"A_1113_MXZ11_O1"	Q 24.2	BOOL	// ASPIRATION FAN TANK 3
"A_1114_MXZ11_O1"	Q 24.3	BOOL	// ASPIRATION FAN TANK 4
"A_1115_MXZ11_O1"	Q 24.4	BOOL	// ASPIRATION FAN TANK 5
"A_1116_MXZ11_O1"	Q 24.5	BOOL	// ASPIRATION FAN TANK 6
"A_1117_MXZ11_O1"	Q 24.6	BOOL	// ASPIRATION FAN TANK 7
"A_1118_MXZ11_O1"	Q 24.7	BOOL	// ASPIRATION FAN TANK 8
"A_1119_MXZ11_O1"	Q 25.0	BOOL	// ASPIRATION FAN TANK 9
"A_1120_MXZ11_O1"	Q 25.1	BOOL	// ASPIRATION FAN TANK 10
"A_1121_MXZ11_O1"	Q 25.2	BOOL	// ASPIRATION FAN TANK 11
"A_1122_MXZ11_O1"	Q 25.3	BOOL	// ASPIRATION FAN TANK 12
"A_1123_MXZ11_O1"	Q 25.4	BOOL	// ASPIRATION FAN TANK 13
"A_1124_MXZ11_O1"	Q 25.5	BOOL	// ASPIRATION FAN TANK 14
"A_1125_MXZ11_O1"	Q 25.6	BOOL	// ASPIRATION FAN TANK 15
"A_1126_MXZ11_O1"	Q 25.7	BOOL	// ASPIRATION FAN TANK 16
"A_1127_MXZ11_O1"	Q 26.0	BOOL	// ASPIRATION FAN TANK 17
"A_1127_MXZ21_O1"	Q 26.1	BOOL	// DISCHARGE SLIDE T17 CLOSED
"A_1127_MXZ21_O2"	Q 26.2	BOOL	// DISCHARGE SLIDE T17 OPENED
"A_1128_MXZ11_O1"	Q 26.3	BOOL	// ASPIRATION FAN TANK 18
"A_1128_MXZ21_O1"	Q 26.4	BOOL	// DISCHARGE SLIDE T18 CLOSED
"A_1128_MXZ21_O2"	Q 26.5	BOOL	// DISCHARGE SLIDE T18 OPENED
"A_1129_MXZ11_O1"	Q 26.6	BOOL	// ASPIRATION FAN TANK 19
"A_1129_MXZ21_O1"	Q 26.7	BOOL	// DISCHARGE SLIDE T19 CLOSED
"A_1129_MXZ21_O2"	Q 27.0	BOOL	// DISCHARGE SLIDE T19 OPENED
"A_1130_MXZ11_O1"	Q 27.1	BOOL	// ASPIRATION FAN TANK 20
"A_1130_MXZ21_O1"	Q 27.2	BOOL	// DISCHARGE SLIDE T20 CLOSED
"A_1130_MXZ21_O2"	Q 27.3	BOOL	// DISCHARGE SLIDE T20 OPENED
"A_1131_MXZ11_O1"	Q 27.4	BOOL	// ASPIRATION FAN TANK 21
"A_1131_MXZ21_O1"	Q 27.5	BOOL	// DISCHARGE SLIDE T21 CLOSED
"A_1131_MXZ21_O2"	Q 27.6	BOOL	// DISCHARGE SLIDE T21 OPENED
"A_1132_MXZ11_O1"	Q 27.7	BOOL	// ASPIRATION FAN TANK 22
"A_1132_MXZ21_O1"	Q 28.0	BOOL	// DISCHARGE SLIDE T22 CLOSED
"A_1132_MXZ21_O2"	Q 28.1	BOOL	// DISCHARGE SLIDE T22 OPENED
"A_1133_MXZ11_O1"	Q 28.2	BOOL	// ASPIRATION FAN TANK 23
"A_1133_MXZ21_O1"	Q 28.3	BOOL	// DISCHARGE SLIDE T23 CLOSED
"A_1133_MXZ21_O2"	Q 28.4	BOOL	// DISCHARGE SLIDE T23 OPENED
"A_1134_MXZ11_O1"	Q 28.5	BOOL	// ASPIRATION FAN TANK 24
"A_1134_MXZ21_O1"	Q 28.6	BOOL	// DISCHARGE SLIDE T24 CLOSED
"A_1134_MXZ21_O2"	Q 28.7	BOOL	// DISCHARGE SLIDE T24 OPENED
"A_1151_MXZ11_O1"	Q 29.0	BOOL	// COMPRESSED AIR GROUP S1-S4
"A_1152_MXZ11_O1"	Q 29.1	BOOL	// COMPRESSED AIR GROUP S5-S8
"A_1153_MXZ11_O1"	Q 29.2	BOOL	// COMPRESSED AIR GROUP S9-S12
"A_1154_MXZ11_O1"	Q 29.3	BOOL	// COMPRESSED AIR GROUP S13-S16
"A_1155_MXZ11_O1"	Q 29.4	BOOL	// COMPRESSED AIR GROUP S17-S20
"A_1156_MXZ11_O1"	Q 29.5	BOOL	// COMPRESSED AIR GROUP S21-S24
"A_1111_QXV42_O2"	Q 32.1	BOOL	// BALL VALVE FRESH-AIR TANK 1
"A_1112_QXV42_O2"	Q 32.3	BOOL	// BALL VALVE FRESH-AIR TANK 2
"A_1113_QXV42_O2"	Q 32.5	BOOL	// BALL VALVE FRESH-AIR TANK 3
"A_1114_QXV42_O2"	Q 32.7	BOOL	// BALL VALVE FRESH-AIR TANK 4
"A_1115_QXV42_O2"	Q 33.1	BOOL	// BALL VALVE FRESH-AIR TANK 5
"A_1116_QXV42_O2"	Q 33.3	BOOL	// BALL VALVE FRESH-AIR TANK 6
"A_1117_QXV42_O2"	Q 33.5	BOOL	// BALL VALVE FRESH-AIR TANK 7
"A_1118_QXV42_O2"	Q 33.7	BOOL	// BALL VALVE FRESH-AIR TANK 8
"A_1119_QXV42_O2"	Q 34.1	BOOL	// BALL VALVE FRESH-AIR TANK 9
"A_1120_QXV42_O2"	Q 34.3	BOOL	// BALL VALVE FRESH-AIR TANK 10
"A_1121_QXV42_O2"	Q 34.5	BOOL	// BALL VALVE FRESH-AIR TANK 11
"A_1122_QXV42_O2"	Q 34.7	BOOL	// BALL VALVE FRESH-AIR TANK 12
"A_1123_QXV42_O2"	Q 44.1	BOOL	// BALL VALVE FRESH-AIR TANK 13
"A_1124_QXV42_O2"	Q 44.3	BOOL	// BALL VALVE FRESH-AIR TANK 14
"A_1125_QXV42_O2"	Q 44.5	BOOL	// BALL VALVE FRESH-AIR TANK 15
"A_1126_QXV42_O2"	Q 44.7	BOOL	// BALL VALVE FRESH-AIR TANK 16
"A_1127_QXV42_O2"	Q 45.1	BOOL	// BALL VALVE FRESH-AIR TANK 17
"A_1128_QXV42_O2"	Q 45.3	BOOL	// BALL VALVE FRESH-AIR TANK 18
"A_1129_QXV42_O2"	Q 45.5	BOOL	// BALL VALVE FRESH-AIR TANK 19
"A_1130_QXV42_O2"	Q 45.7	BOOL	// BALL VALVE FRESH-AIR TANK 20
"A_1131_QXV42_O2"	Q 46.1	BOOL	// BALL VALVE FRESH-AIR TANK 21
"A_1132_QXV42_O2"	Q 46.3	BOOL	// BALL VALVE FRESH-AIR TANK 22
"A_1133_QXV42_O2"	Q 46.5	BOOL	// BALL VALVE FRESH-AIR TANK 23
"A_1134_QXV42_O2"	Q 46.7	BOOL	// BALL VALVE FRESH-AIR TANK 24
"A_1161_MXZ01_O1"	Q 48.0	BOOL	// SLIDE GATE 1 - CO2 OPEN
"A_1161_MXZ01_O2"	Q 48.1	BOOL	// SLIDE GATE 1 - CO2 CLOSE
"A_1162_MXZ01_O1"	Q 48.2	BOOL	// SLIDE GATE 2 - CO2 OPEN
"A_1162_MXZ01_O2"	Q 48.3	BOOL	// SLIDE GATE 2 - CO2 CLOSE
"A_1163_MXZ01_O1"	Q 48.4	BOOL	// SLIDE GATE 3 - CO2 OPEN
"A_1163_MXZ01_O2"	Q 48.5	BOOL	// SLIDE GATE 3 - CO2 CLOSE
"A_1164_MXZ01_O1"	Q 48.6	BOOL	// SLIDE GATE 4 - CO2 OPEN
"A_1164_MXZ01_O2"	Q 48.7	BOOL	// SLIDE GATE 4 - CO2 CLOSE
"A_1165_MXZ01_O1"	Q 49.0	BOOL	// SLIDE GATE 5 - CO2 OPEN
"A_1165_MXZ01_O2"	Q 49.1	BOOL	// SLIDE GATE 5 - CO2 CLOSE
"A_1166_MXZ01_O1"	Q 49.2	BOOL	// SLIDE GATE 6 - CO2 OPEN
"A_1166_MXZ01_O2"	Q 49.3	BOOL	// SLIDE GATE 6 - CO2 CLOSE
"A_1167_MXZ01_O1"	Q 49.4	BOOL	// SLIDE GATE 7 - CO2 OPEN
"A_1167_MXZ01_O2"	Q 49.5	BOOL	// SLIDE GATE 7 - CO2 CLOSE
"A_1168_MXZ01_O1"	Q 49.6	BOOL	// SLIDE GATE 8 - CO2 OPEN
"A_1168_MXZ01_O2"	Q 49.7	BOOL	// SLIDE GATE 8 - CO2 CLOSE
"A_1169_MXZ01_O1"	Q 50.0	BOOL	// SLIDE GATE 9 - CO2 OPEN
"A_1169_MXZ01_O2"	Q 50.1	BOOL	// SLIDE GATE 9 - CO2 CLOSE
"A_1170_MXZ01_O1"	Q 50.2	BOOL	// SLIDE GATE 10-CO2 OPEN
"A_1170_MXZ01_O2"	Q 50.3	BOOL	// SLIDE GATE 10-CO2 CLOSE
"A_1171_MXZ01_O1"	Q 50.4	BOOL	// SLIDE GATE 11-CO2 OPEN
"A_1171_MXZ01_O2"	Q 50.5	BOOL	// SLIDE GATE 11-CO2 CLOSE
"A_1172_MXZ01_O1"	Q 50.6	BOOL	// SLIDE GATE 12-CO2 OPEN
"A_1172_MXZ01_O2"	Q 50.7	BOOL	// SLIDE GATE 12-CO2 CLOSE
"A_1173_MXZ01_O1"	Q 51.0	BOOL	// SLIDE GATE 13-CO2 OPEN
"A_1173_MXZ01_O2"	Q 51.1	BOOL	// SLIDE GATE 13-CO2 CLOSE
"A_1174_MXZ01_O1"	Q 51.2	BOOL	// SLIDE GATE 14-CO2 OPEN
"A_1174_MXZ01_O2"	Q 51.3	BOOL	// SLIDE GATE 14-CO2 CLOSE
"A_1175_MXZ01_O1"	Q 51.4	BOOL	// SLIDE GATE 15-CO2 OPEN
"A_1175_MXZ01_O2"	Q 51.5	BOOL	// SLIDE GATE 15-CO2 CLOSE
"A_1176_MXZ01_O1"	Q 51.6	BOOL	// SLIDE GATE 16-CO2 OPEN
"A_1176_MXZ01_O2"	Q 51.7	BOOL	// SLIDE GATE 16-CO2 CLOSE
"A_1177_MXZ01_O1"	Q 52.0	BOOL	// SLIDE GATE 17-CO2 OPEN
"A_1177_MXZ01_O2"	Q 52.1	BOOL	// SLIDE GATE 17-CO2 CLOSE
"A_1178_MXZ01_O1"	Q 52.2	BOOL	// SLIDE GATE 18-CO2 OPEN
"A_1178_MXZ01_O2"	Q 52.3	BOOL	// SLIDE GATE 18-CO2 CLOSE
"A_1179_MXZ01_O1"	Q 52.4	BOOL	// SLIDE GATE 19-CO2 OPEN
"A_1179_MXZ01_O2"	Q 52.5	BOOL	// SLIDE GATE 19-CO2 CLOSE
"A_1180_MXZ01_O1"	Q 52.6	BOOL	// SLIDE GATE 20-CO2 OPEN
"A_1180_MXZ01_O2"	Q 52.7	BOOL	// SLIDE GATE 20-CO2 CLOSE
"A_1181_MXZ01_O1"	Q 53.0	BOOL	// SLIDE GATE 21-CO2 OPEN
"A_1181_MXZ01_O2"	Q 53.1	BOOL	// SLIDE GATE 21-CO2 CLOSE
"A_1182_MXZ01_O1"	Q 53.2	BOOL	// SLIDE GATE 22-CO2 OPEN
"A_1182_MXZ01_O2"	Q 53.3	BOOL	// SLIDE GATE 22-CO2 CLOSE
"A_1183_MXZ01_O1"	Q 53.4	BOOL	// SLIDE GATE 23-CO2 OPEN
"A_1183_MXZ01_O2"	Q 53.5	BOOL	// SLIDE GATE 23-CO2 CLOSE
"A_1184_MXZ01_O1"	Q 53.6	BOOL	// SLIDE GATE 24-CO2 OPEN
"A_1184_MXZ01_O2"	Q 53.7	BOOL	// SLIDE GATE 24-CO2 CLOSE
"A_1111_MXZ45_O1"	Q 64.0	BOOL	// AERATION-VALVE 1 OPEN
"A_1111_MXZ45_O2"	Q 64.1	BOOL	// AERATION-VALVE 1 CLOSE
"A_1112_MXZ45_O1"	Q 64.2	BOOL	// AERATION-VALVE 2 OPEN
"A_1112_MXZ45_O2"	Q 64.3	BOOL	// AERATION-VALVE 2 CLOSE
"A_1113_MXZ45_O1"	Q 64.4	BOOL	// AERATION-VALVE 3 OPEN
"A_1113_MXZ45_O2"	Q 64.5	BOOL	// AERATION-VALVE 3 CLOSE
"A_1114_MXZ45_O1"	Q 64.6	BOOL	// AERATION-VALVE 4 OPEN
"A_1114_MXZ45_O2"	Q 64.7	BOOL	// AERATION-VALVE 4 CLOSE
"A_1115_MXZ45_O1"	Q 65.0	BOOL	// AERATION-VALVE 5 OPEN
"A_1115_MXZ45_O2"	Q 65.1	BOOL	// AERATION-VALVE 5 CLOSE
"A_1116_MXZ45_O1"	Q 65.2	BOOL	// AERATION-VALVE 6 OPEN
"A_1116_MXZ45_O2"	Q 65.3	BOOL	// AERATION-VALVE 6 CLOSE
"A_1117_MXZ45_O1"	Q 65.4	BOOL	// AERATION-VALVE 7 OPEN
"A_1117_MXZ45_O2"	Q 65.5	BOOL	// AERATION-VALVE 7 CLOSE
"A_1118_MXZ45_O1"	Q 65.6	BOOL	// AERATION-VALVE 8 OPEN
"A_1118_MXZ45_O2"	Q 65.7	BOOL	// AERATION-VALVE 8 CLOSE
"A_2101_MXZ01_O1"	Q 102.0	BOOL	// BELT CONVEYOR
"A_2102_MXZ01_O1"	Q 102.1	BOOL	// CHUTE DRIVE LEFT SIDE
"A_2102_MXZ01_O2"	Q 102.2	BOOL	// CHUTE DRIVE RIGHT SIDE
"A_2111_MXZ61_O1"	Q 103.2	BOOL	// TURNING SCREW DRIVE 1
"A_2111_MXZ62_O1"	Q 103.3	BOOL	// TURNING SCREW DRIVE 2
"A_2111_MXZ63_O1"	Q 103.4	BOOL	// TURNING SCREW DRIVE 3
"A_2111_MXZ64_O1"	Q 103.5	BOOL	// TURNING SCREW DRIVE 4
"A_2111_MXZ65_O1"	Q 103.6	BOOL	// TURNING SCREW DRIVE 5
"A_2111_MXZ66_O1"	Q 103.7	BOOL	// TURNING SCREW DRIVE 6
"A_2111_MXZ67_O1"	Q 104.0	BOOL	// TURNING SCREW DRIVE 7
"A_2111_MXZ68_O1"	Q 104.1	BOOL	// TURNING SCREW DRIVE 8
"A_2111_MXZ69_O1"	Q 104.2	BOOL	// TURNING SCREW DRIVE 9
"A_2111_MXZ70_O1"	Q 104.3	BOOL	// TURNING SCREW DRIVE 10
"A_2111_MXZ71_O1"	Q 104.4	BOOL	// TURNING SCREW DRIVE 11
"A_2111_MXZ72_O1"	Q 104.5	BOOL	// TURNING SCREW DRIVE 12
"A_2111_MXZ73_O1"	Q 104.6	BOOL	// TURNING SCREW DRIVE 13
"A_2115_MXZ11_O1"	Q 108.0	BOOL	// HORIZONTAL SCREW
"A_2115_MXZ15_O1"	Q 108.2	BOOL	// LIFTING SCREW
"A_2115_MXZ21_O1"	Q 108.3	BOOL	// LIFTING DEVICE DOWN
"A_2115_MXZ21_O2"	Q 108.4	BOOL	// LIFTING DEVICE UP
"A_2145_QXV21_O1"	Q 116.0	BOOL	// START COOLING UNIT GERMINATING
"A_2145_QXV31_O1"	Q 116.1	BOOL	// START COOLING UNIT GERMINATING
"A_2101_QXV21_O1"	Q 116.2	BOOL	// BALL VALVE SPRAY WATER OPEN
"A_2116_QXV12_O2"	Q 116.4	BOOL	// BALL VALVE SPRINKING WATER LINE
"A_2131_QXV12_O1"	Q 116.6	BOOL	// BALL VALVE AIR HUMIDIFICATION
"A_2131_QXV22_O1"	Q 116.7	BOOL	// BALL VALVE AIR HUMIDIFICATION
"A_2131_QXV12_O2"	Q 117.2	BOOL	// BALL VALVE VALVE HUMIDIFICATION
"A_2199_PAZ11_O1"	Q 118.0	BOOL	// ALARM HORN MACHINE
"A_2112_QXV12_O2"	Q 140.0	BOOL	// BALL VALVE SPRINKING WATER LINE 1
"A_21_A408Z1_O1"	Q 140.1	BOOL	// RESET ALARM
"A_2112_QXV22_O2"	Q 140.2	BOOL	// BALL VALVE SPRINKING WATER LINE 2
"A_2111_KCL01_O1"	Q 140.4	BOOL	// ALARM FLASHER
"A_2111_KCL01_O2"	Q 140.5	BOOL	// SPARE
"A_2111_MXZ21_O1"	Q 141.0	BOOL	// COUPLING DRIVE
"A_2111_MXZ21_O2"	Q 141.1	BOOL	// COUPLING DRIVE
"A_2111_MXZ25_O1"	Q 141.2	BOOL	// COUPLING DRIVE
"A_2111_MXZ25_O2"	Q 141.3	BOOL	// COUPLING DRIVE
"A_2111_MXZ31_O1"	Q 141.4	BOOL	// COUPLING DRIVE
"A_2111_MXZ31_O2"	Q 141.5	BOOL	// COUPLING DRIVE
"A_2111_MXZ35_O1"	Q 141.6	BOOL	// COUPLING DRIVE
"A_2111_MXZ35_O2"	Q 141.7	BOOL	// COUPLING DRIVE
"A_2115_KCL01_O1"	Q 160.0	BOOL	// BACKWALL LIFTED
"A_2115_KCL01_O2"	Q 160.1	BOOL	// BACKWALL LOWERED
"A_2115_KCL01_O3"	Q 160.2	BOOL	// UNCOUPLED
"A_2115_KCL01_O4"	Q 160.3	BOOL	// COUPLED
"A_2115_KCL01_O5"	Q 160.4	BOOL	// WALL LOCKED
"A_2115_KCL01_O6"	Q 160.5	BOOL	// WALL UNLOCKED
"A_2115_KCL01_O7"	Q 160.6	BOOL	// CLEANING FLAP 1/2
"A_2115_MXZ41_O1"	Q 161.0	BOOL	// COUPLING DRIVE
"A_2115_MXZ41_O2"	Q 161.1	BOOL	// COUPLING DRIVE
"A_2115_MXZ45_O1"	Q 161.2	BOOL	// COUPLING DRIVE
"A_2115_MXZ45_O2"	Q 161.3	BOOL	// COUPLING DRIVE
"A_2150_MXZ01_O1"	Q 164.0	BOOL	// AIR-FLAP 1 OPEN
"A_2150_MXZ01_O2"	Q 164.1	BOOL	// AIR-FLAP 1 CLOSE
"A_2151_MXZ01_O1"	Q 164.4	BOOL	// AIR-FLAP 2 OPEN
"A_2151_MXZ01_O2"	Q 164.5	BOOL	// AIR-FLAP 2 CLOSE
"A_2152_MXZ01_O1"	Q 165.0	BOOL	// AIR-FLAP 3 OPEN
"A_2152_MXZ01_O2"	Q 165.1	BOOL	// AIR-FLAP 3 CLOSE
"A_2154_MXZ01_O1"	Q 165.4	BOOL	// WATER PUMP 1
"A_2155_MXZ01_O1"	Q 165.5	BOOL	// WATER PUMP 2
"A_2160_MXZ01_O1"	Q 165.6	BOOL	// GERM FAN 1
"A_2160_MXZ02_O1"	Q 165.7	BOOL	// GERM FAN 2
"A_2201_MXZ01_O1"	Q 202.0	BOOL	// BELT CONVEYOR
"A_2202_MXZ01_O1"	Q 202.1	BOOL	// CHUTE DRIVE LEFT SIDE
"A_2202_MXZ01_O2"	Q 202.2	BOOL	// CHUTE DRIVE RIGHT SIDE
"A_2211_MXZ61_O1"	Q 203.2	BOOL	// TURNING SCREW DRIVE 1
"A_2211_MXZ62_O1"	Q 203.3	BOOL	// TURNING SCREW DRIVE 2
"A_2211_MXZ63_O1"	Q 203.4	BOOL	// TURNING SCREW DRIVE 3
"A_2211_MXZ64_O1"	Q 203.5	BOOL	// TURNING SCREW DRIVE 4
"A_2211_MXZ65_O1"	Q 203.6	BOOL	// TURNING SCREW DRIVE 5
"A_2211_MXZ66_O1"	Q 203.7	BOOL	// TURNING SCREW DRIVE 6
"A_2211_MXZ67_O1"	Q 204.0	BOOL	// TURNING SCREW DRIVE 7
"A_2211_MXZ68_O1"	Q 204.1	BOOL	// TURNING SCREW DRIVE 8
"A_2211_MXZ69_O1"	Q 204.2	BOOL	// TURNING SCREW DRIVE 9
"A_2211_MXZ70_O1"	Q 204.3	BOOL	// TURNING SCREW DRIVE 10
"A_2211_MXZ71_O1"	Q 204.4	BOOL	// TURNING SCREW DRIVE 11
"A_2211_MXZ72_O1"	Q 204.5	BOOL	// TURNING SCREW DRIVE 12
"A_2211_MXZ73_O1"	Q 204.6	BOOL	// TURNING SCREW DRIVE 13
"A_2215_MXZ11_O1"	Q 208.0	BOOL	// HORIZONTAL SCREW
"A_2215_MXZ15_O1"	Q 208.2	BOOL	// LIFTING SCREW
"A_2215_MXZ21_O1"	Q 208.3	BOOL	// LIFTING DEVICE DOWN
"A_2215_MXZ21_O2"	Q 208.4	BOOL	// LIFTING DEVICE UP
"A_2245_QXV21_O1"	Q 216.0	BOOL	// START COOLING UNIT GERMINATING
"A_2245_QXV31_O1"	Q 216.1	BOOL	// START COOLING UNIT GERMINATING
"A_2201_QXV21_O1"	Q 216.2	BOOL	// BALL VALVE SPRAY WATER OPEN
"A_2216_QXV12_O2"	Q 216.4	BOOL	// BALL VALVE SPRINKING WATER LINE
"A_2231_QXV12_O1"	Q 216.6	BOOL	// BALL VALVE AIR HUMIDIFICATION
"A_2231_QXV22_O1"	Q 216.7	BOOL	// BALL VALVE AIR HUMIDIFICATION
"A_2231_QXV12_O2"	Q 217.2	BOOL	// BALL VALVE VALVE HUMIDIFICATION
"A_2299_PAZ11_O1"	Q 218.0	BOOL	// ALARM HORN MACHINE
"A_2212_QXV12_O2"	Q 240.0	BOOL	// BALL VALVE SPRINKING WATER LINE 1
"A_22_A408Z1_O1"	Q 240.1	BOOL	// RESET ALARM
"A_2212_QXV22_O2"	Q 240.2	BOOL	// BALL VALVE SPRINKING WATER LINE 2
"A_2211_KCL01_O1"	Q 240.4	BOOL	// ALARM FLASHER
"A_2211_KCL01_O2"	Q 240.5	BOOL	// SPARE
"A_2211_MXZ21_O1"	Q 241.0	BOOL	// COUPLING DRIVE
"A_2211_MXZ21_O2"	Q 241.1	BOOL	// COUPLING DRIVE
"A_2211_MXZ25_O1"	Q 241.2	BOOL	// COUPLING DRIVE
"A_2211_MXZ25_O2"	Q 241.3	BOOL	// COUPLING DRIVE
"A_2211_MXZ31_O1"	Q 241.4	BOOL	// COUPLING DRIVE
"A_2211_MXZ31_O2"	Q 241.5	BOOL	// COUPLING DRIVE
"A_2211_MXZ35_O1"	Q 241.6	BOOL	// COUPLING DRIVE
"A_2211_MXZ35_O2"	Q 241.7	BOOL	// COUPLING DRIVE
"A_2215_KCL01_O1"	Q 260.0	BOOL	// BACKWALL LIFTED
"A_2215_KCL01_O2"	Q 260.1	BOOL	// BACKWALL LOWERED
"A_2215_KCL01_O3"	Q 260.2	BOOL	// UNCOUPLED
"A_2215_KCL01_O4"	Q 260.3	BOOL	// COUPLED
"A_2215_KCL01_O5"	Q 260.4	BOOL	// WALL LOCKED
"A_2215_KCL01_O6"	Q 260.5	BOOL	// WALL UNLOCKED
"A_2215_KCL01_O7"	Q 260.6	BOOL	// CLEANING FLAP 1/2
"A_2215_MXZ41_O1"	Q 261.0	BOOL	// COUPLING DRIVE
"A_2215_MXZ41_O2"	Q 261.1	BOOL	// COUPLING DRIVE
"A_2215_MXZ45_O1"	Q 261.2	BOOL	// COUPLING DRIVE
"A_2215_MXZ45_O2"	Q 261.3	BOOL	// COUPLING DRIVE
"A_2250_MXZ01_O1"	Q 264.0	BOOL	// AIR-FLAP 1 OPEN
"A_2250_MXZ01_O2"	Q 264.1	BOOL	// AIR-FLAP 1 CLOSE
"A_2251_MXZ01_O1"	Q 264.4	BOOL	// AIR-FLAP 2 OPEN
"A_2251_MXZ01_O2"	Q 264.5	BOOL	// AIR-FLAP 2 CLOSE
"A_2252_MXZ01_O1"	Q 265.0	BOOL	// AIR-FLAP 3 OPEN
"A_2252_MXZ01_O2"	Q 265.1	BOOL	// AIR-FLAP 3 CLOSE
"A_2254_MXZ01_O1"	Q 265.4	BOOL	// WATER PUMP 1
"A_2255_MXZ01_O1"	Q 265.5	BOOL	// WATER PUMP 2
"A_2260_MXZ01_O1"	Q 265.6	BOOL	// GERM FAN 1
"A_2260_MXZ02_O1"	Q 265.7	BOOL	// GERM FAN 2
"A_2301_MXZ01_O1"	Q 302.0	BOOL	// BELT CONVEYOR
"A_2302_MXZ01_O1"	Q 302.1	BOOL	// CHUTE DRIVE LEFT SIDE
"A_2302_MXZ01_O2"	Q 302.2	BOOL	// CHUTE DRIVE RIGHT SIDE
"A_2311_MXZ61_O1"	Q 303.2	BOOL	// TURNING SCREW DRIVE 1
"A_2311_MXZ62_O1"	Q 303.3	BOOL	// TURNING SCREW DRIVE 2
"A_2311_MXZ63_O1"	Q 303.4	BOOL	// TURNING SCREW DRIVE 3
"A_2311_MXZ64_O1"	Q 303.5	BOOL	// TURNING SCREW DRIVE 4
"A_2311_MXZ65_O1"	Q 303.6	BOOL	// TURNING SCREW DRIVE 5
"A_2311_MXZ66_O1"	Q 303.7	BOOL	// TURNING SCREW DRIVE 6
"A_2311_MXZ67_O1"	Q 304.0	BOOL	// TURNING SCREW DRIVE 7
"A_2311_MXZ68_O1"	Q 304.1	BOOL	// TURNING SCREW DRIVE 8
"A_2311_MXZ69_O1"	Q 304.2	BOOL	// TURNING SCREW DRIVE 9
"A_2311_MXZ70_O1"	Q 304.3	BOOL	// TURNING SCREW DRIVE 10
"A_2311_MXZ71_O1"	Q 304.4	BOOL	// TURNING SCREW DRIVE 11
"A_2311_MXZ72_O1"	Q 304.5	BOOL	// TURNING SCREW DRIVE 12
"A_2311_MXZ73_O1"	Q 304.6	BOOL	// TURNING SCREW DRIVE 13
"A_2315_MXZ11_O1"	Q 308.0	BOOL	// HORIZONTAL SCREW
"A_2315_MXZ15_O1"	Q 308.2	BOOL	// LIFTING SCREW
"A_2315_MXZ21_O1"	Q 308.3	BOOL	// LIFTING DEVICE DOWN
"A_2315_MXZ21_O2"	Q 308.4	BOOL	// LIFTING DEVICE UP
"A_2345_QXV21_O1"	Q 316.0	BOOL	// START COOLING UNIT GERMINATING
"A_2345_QXV31_O1"	Q 316.1	BOOL	// START COOLING UNIT GERMINATING
"A_2301_QXV21_O1"	Q 316.2	BOOL	// BALL VALVE SPRAY WATER OPEN
"A_2316_QXV12_O2"	Q 316.4	BOOL	// BALL VALVE SPRINKING WATER LINE
"A_2331_QXV12_O1"	Q 316.6	BOOL	// BALL VALVE AIR HUMIDIFICATION
"A_2331_QXV22_O1"	Q 316.7	BOOL	// BALL VALVE AIR HUMIDIFICATION
"A_2331_QXV12_O2"	Q 317.2	BOOL	// BALL VALVE VALVE HUMIDIFICATION
"A_2399_PAZ11_O1"	Q 318.0	BOOL	// ALARM HORN MACHINE
"A_2312_QXV12_O2"	Q 340.0	BOOL	// BALL VALVE SPRINKING WATER LINE 1
"A_23_A408Z1_O1"	Q 340.1	BOOL	// RESET ALARM
"A_2312_QXV22_O2"	Q 340.2	BOOL	// BALL VALVE SPRINKING WATER LINE 2
"A_2311_KCL01_O1"	Q 340.4	BOOL	// ALARM FLASHER
"A_2311_KCL01_O2"	Q 340.5	BOOL	// SPARE
"A_2311_MXZ21_O1"	Q 341.0	BOOL	// COUPLING DRIVE
"A_2311_MXZ21_O2"	Q 341.1	BOOL	// COUPLING DRIVE
"A_2311_MXZ25_O1"	Q 341.2	BOOL	// COUPLING DRIVE
"A_2311_MXZ25_O2"	Q 341.3	BOOL	// COUPLING DRIVE
"A_2311_MXZ31_O1"	Q 341.4	BOOL	// COUPLING DRIVE
"A_2311_MXZ31_O2"	Q 341.5	BOOL	// COUPLING DRIVE
"A_2311_MXZ35_O1"	Q 341.6	BOOL	// COUPLING DRIVE
"A_2311_MXZ35_O2"	Q 341.7	BOOL	// COUPLING DRIVE
"A_2315_KCL01_O1"	Q 360.0	BOOL	// BACKWALL LIFTED
"A_2315_KCL01_O2"	Q 360.1	BOOL	// BACKWALL LOWERED
"A_2315_KCL01_O3"	Q 360.2	BOOL	// UNCOUPLED
"A_2315_KCL01_O4"	Q 360.3	BOOL	// COUPLED
"A_2315_KCL01_O5"	Q 360.4	BOOL	// WALL LOCKED
"A_2315_KCL01_O6"	Q 360.5	BOOL	// WALL UNLOCKED
"A_2315_KCL01_O7"	Q 360.6	BOOL	// CLEANING FLAP 1/2
"A_2315_MXZ41_O1"	Q 361.0	BOOL	// COUPLING DRIVE
"A_2315_MXZ41_O2"	Q 361.1	BOOL	// COUPLING DRIVE
"A_2315_MXZ45_O1"	Q 361.2	BOOL	// COUPLING DRIVE
"A_2315_MXZ45_O2"	Q 361.3	BOOL	// COUPLING DRIVE
"A_2350_MXZ01_O1"	Q 364.0	BOOL	// AIR-FLAP 1 OPEN
"A_2350_MXZ01_O2"	Q 364.1	BOOL	// AIR-FLAP 1 CLOSE
"A_2351_MXZ01_O1"	Q 364.4	BOOL	// AIR-FLAP 2 OPEN
"A_2351_MXZ01_O2"	Q 364.5	BOOL	// AIR-FLAP 2 CLOSE
"A_2352_MXZ01_O1"	Q 365.0	BOOL	// AIR-FLAP 3 OPEN
"A_2352_MXZ01_O2"	Q 365.1	BOOL	// AIR-FLAP 3 CLOSE
"A_2354_MXZ01_O1"	Q 365.4	BOOL	// WATER PUMP 1
"A_2355_MXZ01_O1"	Q 365.5	BOOL	// WATER PUMP 2
"A_2360_MXZ01_O1"	Q 365.6	BOOL	// GERM FAN 1
"A_2360_MXZ02_O1"	Q 365.7	BOOL	// GERM FAN 2
"A_2401_MXZ01_O1"	Q 402.0	BOOL	// BELT CONVEYOR
"A_2402_MXZ01_O1"	Q 402.1	BOOL	// CHUTE DRIVE LEFT SIDE
"A_2402_MXZ01_O2"	Q 402.2	BOOL	// CHUTE DRIVE RIGHT SIDE
"A_2411_MXZ61_O1"	Q 403.2	BOOL	// TURNING SCREW DRIVE 1
"A_2411_MXZ62_O1"	Q 403.3	BOOL	// TURNING SCREW DRIVE 2
"A_2411_MXZ63_O1"	Q 403.4	BOOL	// TURNING SCREW DRIVE 3
"A_2411_MXZ64_O1"	Q 403.5	BOOL	// TURNING SCREW DRIVE 4
"A_2411_MXZ65_O1"	Q 403.6	BOOL	// TURNING SCREW DRIVE 5
"A_2411_MXZ66_O1"	Q 403.7	BOOL	// TURNING SCREW DRIVE 6
"A_2411_MXZ67_O1"	Q 404.0	BOOL	// TURNING SCREW DRIVE 7
"A_2411_MXZ68_O1"	Q 404.1	BOOL	// TURNING SCREW DRIVE 8
"A_2411_MXZ69_O1"	Q 404.2	BOOL	// TURNING SCREW DRIVE 9
"A_2411_MXZ70_O1"	Q 404.3	BOOL	// TURNING SCREW DRIVE 10
"A_2411_MXZ71_O1"	Q 404.4	BOOL	// TURNING SCREW DRIVE 11
"A_2411_MXZ72_O1"	Q 404.5	BOOL	// TURNING SCREW DRIVE 12
"A_2411_MXZ73_O1"	Q 404.6	BOOL	// TURNING SCREW DRIVE 13
"A_2415_MXZ11_O1"	Q 408.0	BOOL	// HORIZONTAL SCREW
"A_2415_MXZ15_O1"	Q 408.2	BOOL	// LIFTING SCREW
"A_2415_MXZ21_O1"	Q 408.3	BOOL	// LIFTING DEVICE DOWN
"A_2415_MXZ21_O2"	Q 408.4	BOOL	// LIFTING DEVICE UP
"A_2445_QXV21_O1"	Q 416.0	BOOL	// START COOLING UNIT GERMINATING
"A_2445_QXV31_O1"	Q 416.1	BOOL	// START COOLING UNIT GERMINATING
"A_2401_QXV21_O1"	Q 416.2	BOOL	// BALL VALVE SPRAY WATER OPEN
"A_2416_QXV12_O2"	Q 416.4	BOOL	// BALL VALVE SPRINKING WATER LINE
"A_2431_QXV12_O1"	Q 416.6	BOOL	// BALL VALVE AIR HUMIDIFICATION
"A_2431_QXV22_O1"	Q 416.7	BOOL	// BALL VALVE AIR HUMIDIFICATION
"A_2431_QXV12_O2"	Q 417.2	BOOL	// BALL VALVE VALVE HUMIDIFICATION
"A_2499_PAZ11_O1"	Q 418.0	BOOL	// ALARM HORN MACHINE
"A_2412_QXV12_O2"	Q 440.0	BOOL	// BALL VALVE SPRINKING WATER LINE 1
"A_24_A408Z1_O1"	Q 440.1	BOOL	// RESET ALARM
"A_2412_QXV22_O2"	Q 440.2	BOOL	// BALL VALVE SPRINKING WATER LINE 2
"A_2411_KCL01_O1"	Q 440.4	BOOL	// ALARM FLASHER
"A_2411_KCL01_O2"	Q 440.5	BOOL	// SPARE
"A_2411_MXZ21_O1"	Q 441.0	BOOL	// COUPLING DRIVE
"A_2411_MXZ21_O2"	Q 441.1	BOOL	// COUPLING DRIVE
"A_2411_MXZ25_O1"	Q 441.2	BOOL	// COUPLING DRIVE
"A_2411_MXZ25_O2"	Q 441.3	BOOL	// COUPLING DRIVE
"A_2411_MXZ31_O1"	Q 441.4	BOOL	// COUPLING DRIVE
"A_2411_MXZ31_O2"	Q 441.5	BOOL	// COUPLING DRIVE
"A_2411_MXZ35_O1"	Q 441.6	BOOL	// COUPLING DRIVE
"A_2411_MXZ35_O2"	Q 441.7	BOOL	// COUPLING DRIVE
"A_2415_KCL01_O1"	Q 460.0	BOOL	// BACKWALL LIFTED
"A_2415_KCL01_O2"	Q 460.1	BOOL	// BACKWALL LOWERED
"A_2415_KCL01_O3"	Q 460.2	BOOL	// UNCOUPLED
"A_2415_KCL01_O4"	Q 460.3	BOOL	// COUPLED
"A_2415_KCL01_O5"	Q 460.4	BOOL	// WALL LOCKED
"A_2415_KCL01_O6"	Q 460.5	BOOL	// WALL UNLOCKED
"A_2415_KCL01_O7"	Q 460.6	BOOL	// CLEANING FLAP 1/2
"A_2415_MXZ41_O1"	Q 461.0	BOOL	// COUPLING DRIVE
"A_2415_MXZ41_O2"	Q 461.1	BOOL	// COUPLING DRIVE
"A_2415_MXZ45_O1"	Q 461.2	BOOL	// COUPLING DRIVE
"A_2415_MXZ45_O2"	Q 461.3	BOOL	// COUPLING DRIVE
"A_2450_MXZ01_O1"	Q 464.0	BOOL	// AIR-FLAP 1 OPEN
"A_2450_MXZ01_O2"	Q 464.1	BOOL	// AIR-FLAP 1 CLOSE
"A_2451_MXZ01_O1"	Q 464.4	BOOL	// AIR-FLAP 2 OPEN
"A_2451_MXZ01_O2"	Q 464.5	BOOL	// AIR-FLAP 2 CLOSE
"A_2452_MXZ01_O1"	Q 465.0	BOOL	// AIR-FLAP 3 OPEN
"A_2452_MXZ01_O2"	Q 465.1	BOOL	// AIR-FLAP 3 CLOSE
"A_2454_MXZ01_O1"	Q 465.4	BOOL	// WATER PUMP 1
"A_2455_MXZ01_O1"	Q 465.5	BOOL	// WATER PUMP 2
"A_2460_MXZ01_O1"	Q 465.6	BOOL	// GERM FAN 1
"A_2460_MXZ02_O1"	Q 465.7	BOOL	// GERM FAN 2
"A_2501_MXZ01_O1"	Q 502.0	BOOL	// BELT CONVEYOR
"A_2502_MXZ01_O1"	Q 502.1	BOOL	// CHUTE DRIVE LEFT SIDE
"A_2502_MXZ01_O2"	Q 502.2	BOOL	// CHUTE DRIVE RIGHT SIDE
"A_2511_MXZ61_O1"	Q 503.2	BOOL	// TURNING SCREW DRIVE 1
"A_2511_MXZ62_O1"	Q 503.3	BOOL	// TURNING SCREW DRIVE 2
"A_2511_MXZ63_O1"	Q 503.4	BOOL	// TURNING SCREW DRIVE 3
"A_2511_MXZ64_O1"	Q 503.5	BOOL	// TURNING SCREW DRIVE 4
"A_2511_MXZ65_O1"	Q 503.6	BOOL	// TURNING SCREW DRIVE 5
"A_2511_MXZ66_O1"	Q 503.7	BOOL	// TURNING SCREW DRIVE 6
"A_2511_MXZ67_O1"	Q 504.0	BOOL	// TURNING SCREW DRIVE 7
"A_2511_MXZ68_O1"	Q 504.1	BOOL	// TURNING SCREW DRIVE 8
"A_2511_MXZ69_O1"	Q 504.2	BOOL	// TURNING SCREW DRIVE 9
"A_2511_MXZ70_O1"	Q 504.3	BOOL	// TURNING SCREW DRIVE 10
"A_2511_MXZ71_O1"	Q 504.4	BOOL	// TURNING SCREW DRIVE 11
"A_2511_MXZ72_O1"	Q 504.5	BOOL	// TURNING SCREW DRIVE 12
"A_2511_MXZ73_O1"	Q 504.6	BOOL	// TURNING SCREW DRIVE 13
"A_2515_MXZ11_O1"	Q 508.0	BOOL	// HORIZONTAL SCREW
"A_2515_MXZ15_O1"	Q 508.2	BOOL	// LIFTING SCREW
"A_2515_MXZ21_O1"	Q 508.3	BOOL	// LIFTING DEVICE DOWN
"A_2515_MXZ21_O2"	Q 508.4	BOOL	// LIFTING DEVICE UP
"A_2545_QXV21_O1"	Q 516.0	BOOL	// START COOLING UNIT GERMINATING
"A_2545_QXV31_O1"	Q 516.1	BOOL	// START COOLING UNIT GERMINATING
"A_2501_QXV21_O1"	Q 516.2	BOOL	// BALL VALVE SPRAY WATER OPEN
"A_2516_QXV12_O2"	Q 516.4	BOOL	// BALL VALVE SPRINKING WATER LINE
"A_2531_QXV12_O1"	Q 516.6	BOOL	// BALL VALVE AIR HUMIDIFICATION
"A_2531_QXV22_O1"	Q 516.7	BOOL	// BALL VALVE AIR HUMIDIFICATION
"A_2531_QXV12_O2"	Q 517.2	BOOL	// BALL VALVE VALVE HUMIDIFICATION
"A_2599_PAZ11_O1"	Q 518.0	BOOL	// ALARM HORN MACHINE
"A_2512_QXV12_O2"	Q 540.0	BOOL	// BALL VALVE SPRINKING WATER LINE 1
"A_25_A408Z1_O1"	Q 540.1	BOOL	// RESET ALARM
"A_2512_QXV22_O2"	Q 540.2	BOOL	// BALL VALVE SPRINKING WATER LINE 2
"A_2511_KCL01_O1"	Q 540.4	BOOL	// ALARM FLASHER
"A_2511_KCL01_O2"	Q 540.5	BOOL	// SPARE
"A_2511_MXZ21_O1"	Q 541.0	BOOL	// COUPLING DRIVE
"A_2511_MXZ21_O2"	Q 541.1	BOOL	// COUPLING DRIVE
"A_2511_MXZ25_O1"	Q 541.2	BOOL	// COUPLING DRIVE
"A_2511_MXZ25_O2"	Q 541.3	BOOL	// COUPLING DRIVE
"A_2511_MXZ31_O1"	Q 541.4	BOOL	// COUPLING DRIVE
"A_2511_MXZ31_O2"	Q 541.5	BOOL	// COUPLING DRIVE
"A_2511_MXZ35_O1"	Q 541.6	BOOL	// COUPLING DRIVE
"A_2511_MXZ35_O2"	Q 541.7	BOOL	// COUPLING DRIVE
"A_2515_KCL01_O1"	Q 560.0	BOOL	// BACKWALL LIFTED
"A_2515_KCL01_O2"	Q 560.1	BOOL	// BACKWALL LOWERED
"A_2515_KCL01_O3"	Q 560.2	BOOL	// UNCOUPLED
"A_2515_KCL01_O4"	Q 560.3	BOOL	// COUPLED
"A_2515_KCL01_O5"	Q 560.4	BOOL	// WALL LOCKED
"A_2515_KCL01_O6"	Q 560.5	BOOL	// WALL UNLOCKED
"A_2515_KCL01_O7"	Q 560.6	BOOL	// CLEANING FLAP 1/2
"A_2515_MXZ41_O1"	Q 561.0	BOOL	// COUPLING DRIVE
"A_2515_MXZ41_O2"	Q 561.1	BOOL	// COUPLING DRIVE
"A_2515_MXZ45_O1"	Q 561.2	BOOL	// COUPLING DRIVE
"A_2515_MXZ45_O2"	Q 561.3	BOOL	// COUPLING DRIVE
"A_2550_MXZ01_O1"	Q 564.0	BOOL	// AIR-FLAP 1 OPEN
"A_2550_MXZ01_O2"	Q 564.1	BOOL	// AIR-FLAP 1 CLOSE
"A_2551_MXZ01_O1"	Q 564.4	BOOL	// AIR-FLAP 2 OPEN
"A_2551_MXZ01_O2"	Q 564.5	BOOL	// AIR-FLAP 2 CLOSE
"A_2552_MXZ01_O1"	Q 565.0	BOOL	// AIR-FLAP 3 OPEN
"A_2552_MXZ01_O2"	Q 565.1	BOOL	// AIR-FLAP 3 CLOSE
"A_2554_MXZ01_O1"	Q 565.4	BOOL	// WATER PUMP 1
"A_2555_MXZ01_O1"	Q 565.5	BOOL	// WATER PUMP 2
"A_2560_MXZ01_O1"	Q 565.6	BOOL	// GERM FAN 1
"A_2560_MXZ02_O1"	Q 565.7	BOOL	// GERM FAN 2
"A_2601_MXZ01_O1"	Q 602.0	BOOL	// BELT CONVEYOR
"A_2602_MXZ01_O1"	Q 602.1	BOOL	// CHUTE DRIVE LEFT SIDE
"A_2602_MXZ01_O2"	Q 602.2	BOOL	// CHUTE DRIVE RIGHT SIDE
"A_2611_MXZ61_O1"	Q 603.2	BOOL	// TURNING SCREW DRIVE 1
"A_2611_MXZ62_O1"	Q 603.3	BOOL	// TURNING SCREW DRIVE 2
"A_2611_MXZ63_O1"	Q 603.4	BOOL	// TURNING SCREW DRIVE 3
"A_2611_MXZ64_O1"	Q 603.5	BOOL	// TURNING SCREW DRIVE 4
"A_2611_MXZ65_O1"	Q 603.6	BOOL	// TURNING SCREW DRIVE 5
"A_2611_MXZ66_O1"	Q 603.7	BOOL	// TURNING SCREW DRIVE 6
"A_2611_MXZ67_O1"	Q 604.0	BOOL	// TURNING SCREW DRIVE 7
"A_2611_MXZ68_O1"	Q 604.1	BOOL	// TURNING SCREW DRIVE 8
"A_2611_MXZ69_O1"	Q 604.2	BOOL	// TURNING SCREW DRIVE 9
"A_2611_MXZ70_O1"	Q 604.3	BOOL	// TURNING SCREW DRIVE 10
"A_2611_MXZ71_O1"	Q 604.4	BOOL	// TURNING SCREW DRIVE 11
"A_2611_MXZ72_O1"	Q 604.5	BOOL	// TURNING SCREW DRIVE 12
"A_2611_MXZ73_O1"	Q 604.6	BOOL	// TURNING SCREW DRIVE 13
"A_2615_MXZ11_O1"	Q 608.0	BOOL	// HORIZONTAL SCREW
"A_2615_MXZ15_O1"	Q 608.2	BOOL	// LIFTING SCREW
"A_2615_MXZ21_O1"	Q 608.3	BOOL	// LIFTING DEVICE DOWN
"A_2615_MXZ21_O2"	Q 608.4	BOOL	// LIFTING DEVICE UP
"A_2645_QXV21_O1"	Q 616.0	BOOL	// START COOLING UNIT GERMINATING
"A_2645_QXV31_O1"	Q 616.1	BOOL	// START COOLING UNIT GERMINATING
"A_2601_QXV21_O1"	Q 616.2	BOOL	// BALL VALVE SPRAY WATER OPEN
"A_2616_QXV12_O2"	Q 616.4	BOOL	// BALL VALVE SPRINKING WATER LINE
"A_2631_QXV12_O1"	Q 616.6	BOOL	// BALL VALVE AIR HUMIDIFICATION
"A_2631_QXV22_O1"	Q 616.7	BOOL	// BALL VALVE AIR HUMIDIFICATION
"A_2631_QXV12_O2"	Q 617.2	BOOL	// BALL VALVE VALVE HUMIDIFICATION
"A_2699_PAZ11_O1"	Q 618.0	BOOL	// ALARM HORN MACHINE
"A_2612_QXV12_O2"	Q 640.0	BOOL	// BALL VALVE SPRINKING WATER LINE 1
"A_26_A408Z1_O1"	Q 640.1	BOOL	// RESET ALARM
"A_2612_QXV22_O2"	Q 640.2	BOOL	// BALL VALVE SPRINKING WATER LINE 2
"A_2611_KCL01_O1"	Q 640.4	BOOL	// ALARM FLASHER
"A_2611_KCL01_O2"	Q 640.5	BOOL	// SPARE
"A_2611_MXZ21_O1"	Q 641.0	BOOL	// COUPLING DRIVE
"A_2611_MXZ21_O2"	Q 641.1	BOOL	// COUPLING DRIVE
"A_2611_MXZ25_O1"	Q 641.2	BOOL	// COUPLING DRIVE
"A_2611_MXZ25_O2"	Q 641.3	BOOL	// COUPLING DRIVE
"A_2611_MXZ31_O1"	Q 641.4	BOOL	// COUPLING DRIVE
"A_2611_MXZ31_O2"	Q 641.5	BOOL	// COUPLING DRIVE
"A_2611_MXZ35_O1"	Q 641.6	BOOL	// COUPLING DRIVE
"A_2611_MXZ35_O2"	Q 641.7	BOOL	// COUPLING DRIVE
"A_2615_KCL01_O1"	Q 660.0	BOOL	// BACKWALL LIFTED
"A_2615_KCL01_O2"	Q 660.1	BOOL	// BACKWALL LOWERED
"A_2615_KCL01_O3"	Q 660.2	BOOL	// UNCOUPLED
"A_2615_KCL01_O4"	Q 660.3	BOOL	// COUPLED
"A_2615_KCL01_O5"	Q 660.4	BOOL	// WALL LOCKED
"A_2615_KCL01_O6"	Q 660.5	BOOL	// WALL UNLOCKED
"A_2615_KCL01_O7"	Q 660.6	BOOL	// CLEANING FLAP 1/2
"A_2615_MXZ41_O1"	Q 661.0	BOOL	// COUPLING DRIVE
"A_2615_MXZ41_O2"	Q 661.1	BOOL	// COUPLING DRIVE
"A_2615_MXZ45_O1"	Q 661.2	BOOL	// COUPLING DRIVE
"A_2615_MXZ45_O2"	Q 661.3	BOOL	// COUPLING DRIVE
"A_2650_MXZ01_O1"	Q 664.0	BOOL	// AIR-FLAP 1 OPEN
"A_2650_MXZ01_O2"	Q 664.1	BOOL	// AIR-FLAP 1 CLOSE
"A_2651_MXZ01_O1"	Q 664.4	BOOL	// AIR-FLAP 2 OPEN
"A_2651_MXZ01_O2"	Q 664.5	BOOL	// AIR-FLAP 2 CLOSE
"A_2652_MXZ01_O1"	Q 665.0	BOOL	// AIR-FLAP 3 OPEN
"A_2652_MXZ01_O2"	Q 665.1	BOOL	// AIR-FLAP 3 CLOSE
"A_2654_MXZ01_O1"	Q 665.4	BOOL	// WATER PUMP 1
"A_2655_MXZ01_O1"	Q 665.5	BOOL	// WATER PUMP 2
"A_2660_MXZ01_O1"	Q 665.6	BOOL	// GERM FAN 1
"A_2660_MXZ02_O1"	Q 665.7	BOOL	// GERM FAN 2
"A_2701_MXZ01_O1"	Q 702.0	BOOL	// BELT CONVEYOR
"A_2702_MXZ01_O1"	Q 702.1	BOOL	// CHUTE DRIVE LEFT SIDE
"A_2702_MXZ01_O2"	Q 702.2	BOOL	// CHUTE DRIVE RIGHT SIDE
"A_2711_MXZ61_O1"	Q 703.2	BOOL	// TURNING SCREW DRIVE 1
"A_2711_MXZ62_O1"	Q 703.3	BOOL	// TURNING SCREW DRIVE 2
"A_2711_MXZ63_O1"	Q 703.4	BOOL	// TURNING SCREW DRIVE 3
"A_2711_MXZ64_O1"	Q 703.5	BOOL	// TURNING SCREW DRIVE 4
"A_2711_MXZ65_O1"	Q 703.6	BOOL	// TURNING SCREW DRIVE 5
"A_2711_MXZ66_O1"	Q 703.7	BOOL	// TURNING SCREW DRIVE 6
"A_2711_MXZ67_O1"	Q 704.0	BOOL	// TURNING SCREW DRIVE 7
"A_2711_MXZ68_O1"	Q 704.1	BOOL	// TURNING SCREW DRIVE 8
"A_2711_MXZ69_O1"	Q 704.2	BOOL	// TURNING SCREW DRIVE 9
"A_2711_MXZ70_O1"	Q 704.3	BOOL	// TURNING SCREW DRIVE 10
"A_2711_MXZ71_O1"	Q 704.4	BOOL	// TURNING SCREW DRIVE 11
"A_2711_MXZ72_O1"	Q 704.5	BOOL	// TURNING SCREW DRIVE 12
"A_2711_MXZ73_O1"	Q 704.6	BOOL	// TURNING SCREW DRIVE 13
"A_2715_MXZ11_O1"	Q 708.0	BOOL	// HORIZONTAL SCREW
"A_2715_MXZ15_O1"	Q 708.2	BOOL	// LIFTING SCREW
"A_2715_MXZ21_O1"	Q 708.3	BOOL	// LIFTING DEVICE DOWN
"A_2715_MXZ21_O2"	Q 708.4	BOOL	// LIFTING DEVICE UP
"A_2745_QXV21_O1"	Q 716.0	BOOL	// START COOLING UNIT GERMINATING
"A_2745_QXV31_O1"	Q 716.1	BOOL	// START COOLING UNIT GERMINATING
"A_2701_QXV21_O1"	Q 716.2	BOOL	// BALL VALVE SPRAY WATER OPEN
"A_2716_QXV12_O2"	Q 716.4	BOOL	// BALL VALVE SPRINKING WATER LINE
"A_2731_QXV12_O1"	Q 716.6	BOOL	// BALL VALVE AIR HUMIDIFICATION
"A_2731_QXV22_O1"	Q 716.7	BOOL	// BALL VALVE AIR HUMIDIFICATION
"A_2731_QXV12_O2"	Q 717.2	BOOL	// BALL VALVE VALVE HUMIDIFICATION
"A_2799_PAZ11_O1"	Q 718.0	BOOL	// ALARM HORN MACHINE
"A_2712_QXV12_O2"	Q 740.0	BOOL	// BALL VALVE SPRINKING WATER LINE 1
"A_27_A408Z1_O1"	Q 740.1	BOOL	// RESET ALARM
"A_2712_QXV22_O2"	Q 740.2	BOOL	// BALL VALVE SPRINKING WATER LINE 2
"A_2711_KCL01_O1"	Q 740.4	BOOL	// ALARM FLASHER
"A_2711_KCL01_O2"	Q 740.5	BOOL	// SPARE
"A_2711_MXZ21_O1"	Q 741.0	BOOL	// COUPLING DRIVE
"A_2711_MXZ21_O2"	Q 741.1	BOOL	// COUPLING DRIVE
"A_2711_MXZ25_O1"	Q 741.2	BOOL	// COUPLING DRIVE
"A_2711_MXZ25_O2"	Q 741.3	BOOL	// COUPLING DRIVE
"A_2711_MXZ31_O1"	Q 741.4	BOOL	// COUPLING DRIVE
"A_2711_MXZ31_O2"	Q 741.5	BOOL	// COUPLING DRIVE
"A_2711_MXZ35_O1"	Q 741.6	BOOL	// COUPLING DRIVE
"A_2711_MXZ35_O2"	Q 741.7	BOOL	// COUPLING DRIVE
"A_2715_KCL01_O1"	Q 760.0	BOOL	// BACKWALL LIFTED
"A_2715_KCL01_O2"	Q 760.1	BOOL	// BACKWALL LOWERED
"A_2715_KCL01_O3"	Q 760.2	BOOL	// UNCOUPLED
"A_2715_KCL01_O4"	Q 760.3	BOOL	// COUPLED
"A_2715_KCL01_O5"	Q 760.4	BOOL	// WALL LOCKED
"A_2715_KCL01_O6"	Q 760.5	BOOL	// WALL UNLOCKED
"A_2715_KCL01_O7"	Q 760.6	BOOL	// CLEANING FLAP 1/2
"A_2715_MXZ41_O1"	Q 761.0	BOOL	// COUPLING DRIVE
"A_2715_MXZ41_O2"	Q 761.1	BOOL	// COUPLING DRIVE
"A_2715_MXZ45_O1"	Q 761.2	BOOL	// COUPLING DRIVE
"A_2715_MXZ45_O2"	Q 761.3	BOOL	// COUPLING DRIVE
"A_2750_MXZ01_O1"	Q 764.0	BOOL	// AIR-FLAP 1 OPEN
"A_2750_MXZ01_O2"	Q 764.1	BOOL	// AIR-FLAP 1 CLOSE
"A_2751_MXZ01_O1"	Q 764.4	BOOL	// AIR-FLAP 2 OPEN
"A_2751_MXZ01_O2"	Q 764.5	BOOL	// AIR-FLAP 2 CLOSE
"A_2752_MXZ01_O1"	Q 765.0	BOOL	// AIR-FLAP 3 OPEN
"A_2752_MXZ01_O2"	Q 765.1	BOOL	// AIR-FLAP 3 CLOSE
"A_2754_MXZ01_O1"	Q 765.4	BOOL	// WATER PUMP 1
"A_2755_MXZ01_O1"	Q 765.5	BOOL	// WATER PUMP 2
"A_2760_MXZ01_O1"	Q 765.6	BOOL	// GERM FAN 1
"A_2760_MXZ02_O1"	Q 765.7	BOOL	// GERM FAN 2
"A_2801_MXZ01_O1"	Q 802.0	BOOL	// BELT CONVEYOR
"A_2802_MXZ01_O1"	Q 802.1	BOOL	// CHUTE DRIVE LEFT SIDE
"A_2802_MXZ01_O2"	Q 802.2	BOOL	// CHUTE DRIVE RIGHT SIDE
"A_2811_MXZ61_O1"	Q 803.2	BOOL	// TURNING SCREW DRIVE 1
"A_2811_MXZ62_O1"	Q 803.3	BOOL	// TURNING SCREW DRIVE 2
"A_2811_MXZ63_O1"	Q 803.4	BOOL	// TURNING SCREW DRIVE 3
"A_2811_MXZ64_O1"	Q 803.5	BOOL	// TURNING SCREW DRIVE 4
"A_2811_MXZ65_O1"	Q 803.6	BOOL	// TURNING SCREW DRIVE 5
"A_2811_MXZ66_O1"	Q 803.7	BOOL	// TURNING SCREW DRIVE 6
"A_2811_MXZ67_O1"	Q 804.0	BOOL	// TURNING SCREW DRIVE 7
"A_2811_MXZ68_O1"	Q 804.1	BOOL	// TURNING SCREW DRIVE 8
"A_2811_MXZ69_O1"	Q 804.2	BOOL	// TURNING SCREW DRIVE 9
"A_2811_MXZ70_O1"	Q 804.3	BOOL	// TURNING SCREW DRIVE 10
"A_2811_MXZ71_O1"	Q 804.4	BOOL	// TURNING SCREW DRIVE 11
"A_2811_MXZ72_O1"	Q 804.5	BOOL	// TURNING SCREW DRIVE 12
"A_2811_MXZ73_O1"	Q 804.6	BOOL	// TURNING SCREW DRIVE 13
"A_2815_MXZ11_O1"	Q 808.0	BOOL	// HORIZONTAL SCREW
"A_2815_MXZ15_O1"	Q 808.2	BOOL	// LIFTING SCREW
"A_2815_MXZ21_O1"	Q 808.3	BOOL	// LIFTING DEVICE DOWN
"A_2815_MXZ21_O2"	Q 808.4	BOOL	// LIFTING DEVICE UP
"A_2845_QXV21_O1"	Q 816.0	BOOL	// START COOLING UNIT GERMINATING
"A_2845_QXV31_O1"	Q 816.1	BOOL	// START COOLING UNIT GERMINATING
"A_2801_QXV21_O1"	Q 816.2	BOOL	// BALL VALVE SPRAY WATER OPEN
"A_2816_QXV12_O2"	Q 816.4	BOOL	// BALL VALVE SPRINKING WATER LINE
"A_2831_QXV12_O1"	Q 816.6	BOOL	// BALL VALVE AIR HUMIDIFICATION
"A_2831_QXV22_O1"	Q 816.7	BOOL	// BALL VALVE AIR HUMIDIFICATION
"A_2831_QXV12_O2"	Q 817.2	BOOL	// BALL VALVE VALVE HUMIDIFICATION
"A_2899_PAZ11_O1"	Q 818.0	BOOL	// ALARM HORN MACHINE
"A_2812_QXV12_O2"	Q 840.0	BOOL	// BALL VALVE SPRINKING WATER LINE 1
"A_28_A408Z1_O1"	Q 840.1	BOOL	// RESET ALARM
"A_2812_QXV22_O2"	Q 840.2	BOOL	// BALL VALVE SPRINKING WATER LINE 2
"A_2811_KCL01_O1"	Q 840.4	BOOL	// ALARM FLASHER
"A_2811_KCL01_O2"	Q 840.5	BOOL	// SPARE
"A_2811_MXZ21_O1"	Q 841.0	BOOL	// COUPLING DRIVE
"A_2811_MXZ21_O2"	Q 841.1	BOOL	// COUPLING DRIVE
"A_2811_MXZ25_O1"	Q 841.2	BOOL	// COUPLING DRIVE
"A_2811_MXZ25_O2"	Q 841.3	BOOL	// COUPLING DRIVE
"A_2811_MXZ31_O1"	Q 841.4	BOOL	// COUPLING DRIVE
"A_2811_MXZ31_O2"	Q 841.5	BOOL	// COUPLING DRIVE
"A_2811_MXZ35_O1"	Q 841.6	BOOL	// COUPLING DRIVE
"A_2811_MXZ35_O2"	Q 841.7	BOOL	// COUPLING DRIVE
"A_2815_KCL01_O1"	Q 860.0	BOOL	// BACKWALL LIFTED
"A_2815_KCL01_O2"	Q 860.1	BOOL	// BACKWALL LOWERED
"A_2815_KCL01_O3"	Q 860.2	BOOL	// UNCOUPLED
"A_2815_KCL01_O4"	Q 860.3	BOOL	// COUPLED
"A_2815_KCL01_O5"	Q 860.4	BOOL	// WALL LOCKED
"A_2815_KCL01_O6"	Q 860.5	BOOL	// WALL UNLOCKED
"A_2815_KCL01_O7"	Q 860.6	BOOL	// CLEANING FLAP 1/2
"A_2815_MXZ41_O1"	Q 861.0	BOOL	// COUPLING DRIVE
"A_2815_MXZ41_O2"	Q 861.1	BOOL	// COUPLING DRIVE
"A_2815_MXZ45_O1"	Q 861.2	BOOL	// COUPLING DRIVE
"A_2815_MXZ45_O2"	Q 861.3	BOOL	// COUPLING DRIVE
"A_2850_MXZ01_O1"	Q 864.0	BOOL	// AIR-FLAP 1 OPEN
"A_2850_MXZ01_O2"	Q 864.1	BOOL	// AIR-FLAP 1 CLOSE
"A_2851_MXZ01_O1"	Q 864.4	BOOL	// AIR-FLAP 2 OPEN
"A_2851_MXZ01_O2"	Q 864.5	BOOL	// AIR-FLAP 2 CLOSE
"A_2852_MXZ01_O1"	Q 865.0	BOOL	// AIR-FLAP 3 OPEN
"A_2852_MXZ01_O2"	Q 865.1	BOOL	// AIR-FLAP 3 CLOSE
"A_2854_MXZ01_O1"	Q 865.4	BOOL	// WATER PUMP 1
"A_2855_MXZ01_O1"	Q 865.5	BOOL	// WATER PUMP 2
"A_2860_MXZ01_O1"	Q 865.6	BOOL	// GERM FAN 1
"A_2860_MXZ02_O1"	Q 865.7	BOOL	// GERM FAN 2
"A_3111_MXZ11_O1"	Q 900.0	BOOL	// UN-/LOADING SCREW DISCHARGE
"A_3111_MXZ21_O1"	Q 900.1	BOOL	// LIFTING DRIVE 1 INSIDE LOWERING
"A_3111_MXZ21_O2"	Q 900.2	BOOL	// LIFTING DRIVE 1 INSIDE LIFTING
"A_3111_MXZ31_O1"	Q 900.3	BOOL	// LIFTING DRIVE 2 OUTSIDE LOWERING
"A_3111_MXZ31_O2"	Q 900.4	BOOL	// LIFTING DRIVE 2 OUTSIDE LIFTING
"A_3111_MXZ41_O1"	Q 900.5	BOOL	// TRAVELING DRIVE
"A_3115_MXZ11_O1"	Q 900.6	BOOL	// DISCHARGE FLAP CLOSE
"A_3115_MXZ11_O2"	Q 900.7	BOOL	// DISCHARGE FLAP OPEN
"A_3135_MXZ11_O1"	Q 901.0	BOOL	// LOUVER RECYCLE AIR 1 CLOSE
"A_3135_MXZ11_O2"	Q 901.1	BOOL	// LOUVER RECYCLE AIR 1 OPEN
"A_3136_MXZ11_O1"	Q 901.2	BOOL	// LOUVER RECYCLE AIR 2 CLOSE
"A_3136_MXZ11_O2"	Q 901.3	BOOL	// LOUVER RECYCLE AIR 2 OPEN
"A_3140_MXZ11_O1"	Q 901.4	BOOL	// LOUVER RECYCLE AIR 1 CLOSE
"A_3140_MXZ11_O2"	Q 901.5	BOOL	// LOUVER RECYCLE AIR 1 OPEN
"A_3141_MXZ11_O1"	Q 901.6	BOOL	// LOUVER RECYCLE AIR 2 CLOSE
"A_3141_MXZ11_O2"	Q 901.7	BOOL	// LOUVER RECYCLE AIR 2 OPEN
"A_3145_MXZ11_O1"	Q 902.0	BOOL	// LOUVER WITHERING AIR 1 CLOSE
"A_3145_MXZ11_O2"	Q 902.1	BOOL	// LOUVER WITHERING AIR 1 OPEN
"A_3146_MXZ11_O1"	Q 902.2	BOOL	// LOUVER WITHERING AIR 2 CLOSE
"A_3146_MXZ11_O2"	Q 902.3	BOOL	// LOUVER WITHERING AIR 2 OPEN
"A_3150_MXZ11_O1"	Q 902.4	BOOL	// LOUVER FRESH AIR 1 CLOSE
"A_3150_MXZ11_O2"	Q 902.5	BOOL	// LOUVER FRESH AIR 1 OPEN
"A_3151_MXZ11_O1"	Q 902.6	BOOL	// LOUVER FRESH AIR 2 CLOSE
"A_3151_MXZ11_O2"	Q 902.7	BOOL	// LOUVER FRESH AIR 2 OPEN
"A_3152_MXZ11_O1"	Q 903.0	BOOL	// LOUVER FRESH AIR 3 CLOSE
"A_3152_MXZ11_O2"	Q 903.1	BOOL	// LOUVER FRESH AIR 3 OPEN
"A_3153_MXZ11_O1"	Q 903.2	BOOL	// LOUVER FRESH AIR 4 CLOSE
"A_3153_MXZ11_O2"	Q 903.3	BOOL	// LOUVER FRESH AIR 4 OPEN
"A_3158_MXZ11_O1"	Q 903.4	BOOL	// LOUVER AIR HEATER 1 CLOSE
"A_3158_MXZ11_O2"	Q 903.5	BOOL	// LOUVER AIR HEATER 1 OPEN
"A_3159_MXZ11_O1"	Q 903.6	BOOL	// LOUVER AIR HEATER 2 CLOSE
"A_3159_MXZ11_O2"	Q 903.7	BOOL	// LOUVER AIR HEATER 2 OPEN
"A_3101_MXZ01_O1"	Q 904.0	BOOL	// OUTLET FLAP DRIVE CLOSE
"A_3101_MXZ01_O2"	Q 904.1	BOOL	// OUTLET FLAP DRIVE OPEN
"A_3125_MXZ02_O1"	Q 904.2	BOOL	// GETRIEBEÖLPUMPE FAN 1
"A_3126_MXZ02_O1"	Q 904.3	BOOL	// GETRIEBEÖLPUMPE FAN 2
"A_3199_PAZ11_O1"	Q 924.0	BOOL	// ALARM HORN
"A_3161_KCL11_O1"	Q 924.2	BOOL	// BURNER 1 MAIN FAN RUNNING
"A_3161_KCL11_O2"	Q 924.3	BOOL	// BURNER 1 EXTERAL ON
"A_3161_KCL12_O1"	Q 924.4	BOOL	// BURNER 2 MAIN FAN RUNNING
"A_3161_KCL12_O2"	Q 924.5	BOOL	// BURNER 2 EXTERAL ON
"A_3211_MXZ11_O1"	Q 1000.0	BOOL	// UN-/LOADING SCREW DISCHARGE
"A_3211_MXZ21_O1"	Q 1000.1	BOOL	// LIFTING DRIVE 1 INSIDE LOWERING
"A_3211_MXZ21_O2"	Q 1000.2	BOOL	// LIFTING DRIVE 1 INSIDE LIFTING
"A_3211_MXZ31_O1"	Q 1000.3	BOOL	// LIFTING DRIVE 2 OUTSIDE LOWERING
"A_3211_MXZ31_O2"	Q 1000.4	BOOL	// LIFTING DRIVE 2 OUTSIDE LIFTING
"A_3211_MXZ41_O1"	Q 1000.5	BOOL	// TRAVELING DRIVE
"A_3215_MXZ11_O1"	Q 1000.6	BOOL	// DISCHARGE FLAP CLOSE
"A_3215_MXZ11_O2"	Q 1000.7	BOOL	// DISCHARGE FLAP OPEN
"A_3235_MXZ11_O1"	Q 1001.0	BOOL	// LOUVER RECYCLE AIR 1 CLOSE
"A_3235_MXZ11_O2"	Q 1001.1	BOOL	// LOUVER RECYCLE AIR 1 OPEN
"A_3236_MXZ11_O1"	Q 1001.2	BOOL	// LOUVER RECYCLE AIR 2 CLOSE
"A_3236_MXZ11_O2"	Q 1001.3	BOOL	// LOUVER RECYCLE AIR 2 OPEN
"A_3240_MXZ11_O1"	Q 1001.4	BOOL	// LOUVER RECYCLE AIR 1 CLOSE
"A_3240_MXZ11_O2"	Q 1001.5	BOOL	// LOUVER RECYCLE AIR 1 OPEN
"A_3241_MXZ11_O1"	Q 1001.6	BOOL	// LOUVER RECYCLE AIR 2 CLOSE
"A_3241_MXZ11_O2"	Q 1001.7	BOOL	// LOUVER RECYCLE AIR 2 OPEN
"A_3245_MXZ11_O1"	Q 1002.0	BOOL	// LOUVER WITHERING AIR 1 CLOSE
"A_3245_MXZ11_O2"	Q 1002.1	BOOL	// LOUVER WITHERING AIR 1 OPEN
"A_3246_MXZ11_O1"	Q 1002.2	BOOL	// LOUVER WITHERING AIR 2 CLOSE
"A_3246_MXZ11_O2"	Q 1002.3	BOOL	// LOUVER WITHERING AIR 2 OPEN
"A_3250_MXZ11_O1"	Q 1002.4	BOOL	// LOUVER FRESH AIR 1 CLOSE
"A_3250_MXZ11_O2"	Q 1002.5	BOOL	// LOUVER FRESH AIR 1 OPEN
"A_3251_MXZ11_O1"	Q 1002.6	BOOL	// LOUVER FRESH AIR 2 CLOSE
"A_3251_MXZ11_O2"	Q 1002.7	BOOL	// LOUVER FRESH AIR 2 OPEN
"A_3252_MXZ11_O1"	Q 1003.0	BOOL	// LOUVER FRESH AIR 3 CLOSE
"A_3252_MXZ11_O2"	Q 1003.1	BOOL	// LOUVER FRESH AIR 3 OPEN
"A_3253_MXZ11_O1"	Q 1003.2	BOOL	// LOUVER FRESH AIR 4 CLOSE
"A_3253_MXZ11_O2"	Q 1003.3	BOOL	// LOUVER FRESH AIR 4 OPEN
"A_3258_MXZ11_O1"	Q 1003.4	BOOL	// LOUVER AIR HEATER 1 CLOSE
"A_3258_MXZ11_O2"	Q 1003.5	BOOL	// LOUVER AIR HEATER 1 OPEN
"A_3259_MXZ11_O1"	Q 1003.6	BOOL	// LOUVER AIR HEATER 2 CLOSE
"A_3259_MXZ11_O2"	Q 1003.7	BOOL	// LOUVER AIR HEATER 2 OPEN
"A_3201_MXZ01_O1"	Q 1004.0	BOOL	// OUTLET FLAP DRIVE CLOSE
"A_3201_MXZ01_O2"	Q 1004.1	BOOL	// OUTLET FLAP DRIVE OPEN
"A_3225_MXZ02_O1"	Q 1004.2	BOOL	// GETRIEBEÖLPUMPE FAN 1
"A_3226_MXZ02_O1"	Q 1004.3	BOOL	// GETRIEBEÖLPUMPE FAN 1
"A_3299_PAZ11_O1"	Q 1024.0	BOOL	// ALARM HORN
"A_3261_KCL11_O1"	Q 1024.2	BOOL	// BURNER 3 MAIN FAN RUNNING
"A_3261_KCL11_O2"	Q 1024.3	BOOL	// BURNER 3 EXTERAL ON
"A_1911_MXZ01_O1"	Q 1102.0	BOOL	// BELT CONVEYOR
"A_1915_MXZ01_O1"	Q 1102.1	BOOL	// BELT CONVEYOR
"A_1921_MXZ01_O1"	Q 1102.2	BOOL	// BELT CONVEYOR
"A_1931_MXZ01_O1"	Q 1102.3	BOOL	// BELT CONVEYOR
"A_1941_MXZ01_O1"	Q 1102.4	BOOL	// BELT CONVEYOR
"A_1942_MXZ01_O3"	Q 1102.5	BOOL	// CHUTE DRIVE LOW ROTARY SPEED
"A_1942_MXZ01_O1"	Q 1102.6	BOOL	// CHUTE DRIVE LEFT SIDE
"A_1942_MXZ01_O2"	Q 1102.7	BOOL	// CHUTE DRIVE RIGHT SIDE
"A_1999_PAZ11_O1"	Q 1104.0	BOOL	// ALARM HORN
"A_1911_QXV31_O1"	Q 1108.0	BOOL	// BALL VALVE SPRAY WATER OPEN
"A_1915_QXV31_O1"	Q 1108.1	BOOL	// BALL VALVE SPRAY WATER OPEN
"A_1921_QXV31_O1"	Q 1108.2	BOOL	// BALL VALVE SPRAY WATER OPEN
"A_1931_QXV31_O1"	Q 1108.3	BOOL	// BALL VALVE SPRAY WATER OPEN
"A_1941_QXV31_O1"	Q 1108.4	BOOL	// BALL VALVE SPRAY WATER OPEN
"A_2911_MXZ01_O1"	Q 1118.0	BOOL	// BELT CONVEYOR
"A_2914_MXZ01_O1"	Q 1118.1	BOOL	// BELT CONVEYOR
"A_2917_MXZ01_O1"	Q 1118.2	BOOL	// BELT CONVEYOR
"A_2920_MXZ01_O1"	Q 1118.3	BOOL	// BELT CONVEYOR
"A_2923_MXZ01_O1"	Q 1118.4	BOOL	// BELT CONVEYOR
"A_2926_MXZ01_O1"	Q 1118.5	BOOL	// BELT CONVEYOR
"A_2929_MXZ01_O1"	Q 1118.6	BOOL	// BELT CONVEYOR
"A_2932_MXZ01_02_O1"	Q 1119.1	BOOL	// BELT CONVEYOR DRIVE 1/2
"A_2935_MXZ01_O1"	Q 1119.2	BOOL	// BELT CONVEYOR RIGHT
"A_2935_MXZ01_O2"	Q 1119.3	BOOL	// BELT CONVEYOR LEFT
"A_2999_PAZ11_O1"	Q 1120.0	BOOL	// ALARM HORN
"A_2911_QXV31_O1"	Q 1124.0	BOOL	// BALL VALVE SPRAY WATER OPEN
"A_2914_QXV31_O1"	Q 1124.1	BOOL	// BALL VALVE SPRAY WATER OPEN
"A_2917_QXV31_O1"	Q 1124.2	BOOL	// BALL VALVE SPRAY WATER OPEN
"A_2920_QXV31_O1"	Q 1124.3	BOOL	// BALL VALVE SPRAY WATER OPEN
"A_2923_QXV31_O1"	Q 1124.4	BOOL	// BALL VALVE SPRAY WATER OPEN
"A_2926_QXV31_O1"	Q 1124.5	BOOL	// BALL VALVE SPRAY WATER OPEN
"A_2935_QXV31_O1"	Q 1124.6	BOOL	// BALL VALVE SPRAY WATER OPEN
"A_2935_QXV41_O1"	Q 1124.7	BOOL	// BALL VALVE SPRAY WATER OPEN
"A_2929_QXV31_O1"	Q 1125.0	BOOL	// BALL VALVE SPRAY WATER OPEN
"A_3946_MXZ01_O1"	Q 1132.4	BOOL	// FLAP BOX 3946 - CMD TO LN
"A_3946_MXZ01_O2"	Q 1132.6	BOOL	// FLAP BOX 3946 - CMD TO HN
"A_3911_MXZ01_O1"	Q 1134.0	BOOL	// CHAIN CONVEYOR
"A_3912_MXZ01_O1"	Q 1134.1	BOOL	// OUTLET FLAP DRIVE CLOSE
"A_3912_MXZ01_O2"	Q 1134.2	BOOL	// OUTLET FLAP DRIVE OPEN
"A_3921_MXZ01_O1"	Q 1134.4	BOOL	// CHAIN CONVEYOR
"A_3922_MXZ01_O1"	Q 1134.5	BOOL	// OUTLET FLAP DRIVE CLOSE
"A_3922_MXZ01_O2"	Q 1134.6	BOOL	// OUTLET FLAP DRIVE OPEN
"A_3930_MXZ01_O1"	Q 1135.0	BOOL	// ELEVATOR
"A_3935_MXZ01_O1"	Q 1135.2	BOOL	// FLAP BOX DRIVE RIGHT SIDE
"A_3935_MXZ01_O2"	Q 1135.3	BOOL	// FLAP BOX DRIVE LEFT SIDE
"A_3938_MXZ01_O1"	Q 1135.4	BOOL	// BELT CONVEYOR
"A_3945_MXZ01_O1"	Q 1135.5	BOOL	// ELEVATOR
"A_3952_MXZ01_O1"	Q 1135.6	BOOL	// DISCHARGER DMBG DRIVE
"A_3955_MXZ01_O1"	Q 1135.7	BOOL	// SCREW CONVEYOR DRIVE
"A_3952_XCJ20_O1"	Q 1136.0	BOOL	// VALVE DMBG CLOSE
"A_3952_XCJ20_O2"	Q 1136.1	BOOL	// VALVE DMBG OPEN
"A_3952_XCJ20_O3"	Q 1136.2	BOOL	// VALVE DMBG CLOSE
"A_3952_XCJ20_O4"	Q 1136.3	BOOL	// VALVE DMBG OPEN
"A_3960_MXZ01_O1"	Q 1136.4	BOOL	// FAN DRIVE
"A_3965_MXZ01_O1"	Q 1136.5	BOOL	// AIRLOCK
"A_3970_MXZ01_O1"	Q 1136.6	BOOL	// AIRLOCK
"A_3999_PAZ11_O1"	Q 1137.0	BOOL	// ALARM HORN
"A_3956_KCL01_O2"	Q 1140.4	BOOL	// LIGHT CUSTOMER ON
"A_3956_KCL01_O3"	Q 1140.5	BOOL	// LIGHT CUSTOMER OFF
"A_3956_KCL01_O1"	Q 1140.6	BOOL	// TURN ON EXCISTING DEGERMINATING SYSTEM
"A_6105_MXZ01_O1"	Q 1152.0	BOOL	// ELEVATOR 6105 - START
"A_6106_MXZ01_O1"	Q 1152.1	BOOL	// SCREW CONV. 6106 - START
"A_6107_MXZ01_O1"	Q 1152.2	BOOL	// OUTLET SLIDE 6107 - CLOSE
"A_6107_MXZ01_O2"	Q 1152.3	BOOL	// OUTLET SLIDE 6107 - OPEN
"A_6108_MXZ01_O1"	Q 1152.4	BOOL	// OUTLET SLIDE 6108 - CLOSE
"A_6108_MXZ01_O2"	Q 1152.5	BOOL	// OUTLET SLIDE 6108 - OPEN
"A_6109_MXZ01_O1"	Q 1152.6	BOOL	// ROUTLET SCREW 6109 - START
"A_6110_MXZ01_O1"	Q 1152.7	BOOL	// ROUTLET SCREW 6110 - START
"A_6111_MXZ01_O1"	Q 1153.0	BOOL	// SIEVE DRIVE 6111 - START
"A_6112_MXZ01_O1"	Q 1153.1	BOOL	// SIEVE DRIVE 6112 - START
"A_6113_MXZ01_O1"	Q 1153.2	BOOL	// CHAIN CONV. 6113 - START
"A_6114_MXZ01_O1"	Q 1153.4	BOOL	// OUTLET SLIDE 6114 - CLOSE
"A_6114_MXZ01_O2"	Q 1153.5	BOOL	// OUTLET SLIDE 6114 - OPEN
"A_6115_MXZ01_O1"	Q 1153.6	BOOL	// OUTLET SLIDE 6115 - CLOSE
"A_6115_MXZ01_O2"	Q 1153.7	BOOL	// OUTLET SLIDE 6115 - OPEN
"A_6116_MXZ01_O1"	Q 1154.0	BOOL	// OUTLET SLIDE 6116 - CLOSE
"A_6116_MXZ01_O2"	Q 1154.1	BOOL	// OUTLET SLIDE 6116 - OPEN
"A_6117_MXZ01_O1"	Q 1154.2	BOOL	// OUTLET SLIDE 6117 - CLOSE
"A_6117_MXZ01_O2"	Q 1154.3	BOOL	// OUTLET SLIDE 6117 - OPEN
"A_6118_MXZ01_O1"	Q 1154.4	BOOL	// CHAIN CONV. 6118 - START
"A_6119_MXZ01_O1"	Q 1154.6	BOOL	// OUTLET SLIDE 6119 - CLOSE
"A_6119_MXZ01_O2"	Q 1154.7	BOOL	// OUTLET SLIDE 6119 - OPEN
"A_6120_MXZ01_O1"	Q 1155.0	BOOL	// OUTLET SLIDE 6120 - CLOSE
"A_6120_MXZ01_O2"	Q 1155.1	BOOL	// OUTLET SLIDE 6120 - OPEN
"A_6121_MXZ01_O1"	Q 1155.2	BOOL	// CHAIN CONV. 6121 - START
"A_6151_MXZ01_O1"	Q 1155.4	BOOL	// OUTLET SLIDE 6151 - CLOSE
"A_6151_MXZ01_O2"	Q 1155.5	BOOL	// OUTLET SLIDE 6151 - OPEN
"A_6152_MXZ01_O1"	Q 1155.6	BOOL	// OUTLET SLIDE 6152 - CLOSE
"A_6152_MXZ01_O2"	Q 1155.7	BOOL	// OUTLET SLIDE 6152 - OPEN
"A_6153_MXZ01_O1"	Q 1156.0	BOOL	// OUTLET SLIDE 6153 - CLOSE
"A_6153_MXZ01_O2"	Q 1156.1	BOOL	// OUTLET SLIDE 6153 - OPEN
"A_6154_MXZ01_O1"	Q 1156.2	BOOL	// OUTLET SLIDE 6154 - CLOSE
"A_6154_MXZ01_O2"	Q 1156.3	BOOL	// OUTLET SLIDE 6154 - OPEN
"A_6155_MXZ01_O1"	Q 1156.4	BOOL	// OUTLET SLIDE 6155 - CLOSE
"A_6155_MXZ01_O2"	Q 1156.5	BOOL	// OUTLET SLIDE 6155 - OPEN
"A_6156_MXZ01_O1"	Q 1156.6	BOOL	// OUTLET SLIDE 6156 - CLOSE
"A_6156_MXZ01_O2"	Q 1156.7	BOOL	// OUTLET SLIDE 6156 - OPEN
"A_6157_MXZ01_O1"	Q 1157.0	BOOL	// OUTLET SLIDE 6157 - CLOSE
"A_6157_MXZ01_O2"	Q 1157.1	BOOL	// OUTLET SLIDE 6157 - OPEN
"A_6161_MXZ01_O1"	Q 1157.2	BOOL	// CHAIN CONV. 6161 - START
"A_6162_MXZ01_O1"	Q 1157.3	BOOL	// CHAIN CONV. 6162 - START
"A_6163_MXZ01_O1"	Q 1157.4	BOOL	// ELEVATOR 6163 - START
"A_6164_MXZ01_O1"	Q 1157.5	BOOL	// SCREW CONV. 6164 - START
"A_6167_MXZ01_O1"	Q 1157.6	BOOL	// SAMPLER 6167 - START
"A_6183_MXZ01_O1"	Q 1157.7	BOOL	// AIRLOCK 6183 - START
"A_6184_MXZ01_O1"	Q 1158.0	BOOL	// ASPIRATIN FAN 6184 - START
"A_6118_KFC10_O2"	Q 1164.0	BOOL	// CONTROL - MAIN FAN STOPPED
"A_6151_KLC01_O1"	Q 1178.0	BOOL	// SIGNAL LAMP OUTLET SLIDE  BIN 198 - OPENED
"A_6151_KLC01_O2"	Q 1178.1	BOOL	// SIGNAL LAMP OUTLET SLIDE  BIN 198 - CLOSED
"A_6151_KLC01_O3"	Q 1178.2	BOOL	// SIGNAL LAMP OUTLET SLIDE  BIN 198 - FAILURE
"A_6152_KLC01_O1"	Q 1178.4	BOOL	// SIGNAL LAMP OUTLET SLIDE  BIN 197 - OPENED
"A_6152_KLC01_O2"	Q 1178.5	BOOL	// SIGNAL LAMP OUTLET SLIDE  BIN 197 - CLOSED
"A_6152_KLC01_O3"	Q 1178.6	BOOL	// SIGNAL LAMP OUTLET SLIDE  BIN 197 - FAILURE
"A_6153_KLC01_O1"	Q 1179.0	BOOL	// SIGNAL LAMP OUTLET SLIDE  BIN 195 - OPENED
"A_6153_KLC01_O2"	Q 1179.1	BOOL	// SIGNAL LAMP OUTLET SLIDE  BIN 195 - CLOSED
"A_6153_KLC01_O3"	Q 1179.2	BOOL	// SIGNAL LAMP OUTLET SLIDE  BIN 195 - FAILURE
"A_6118_KFC10_O1"	Q 1180.0	BOOL	// MVRU FILTER CONTROL - RELEASE
"A_C41_O1"	Q 1180.4	BOOL	// INTERFACE EXP1 - SIGNAL 1
"A_C41_O2"	Q 1180.5	BOOL	// INTERFACE EXP1 - SIGNAL 2
"A_C41_O3"	Q 1180.6	BOOL	// INTERFACE EXP1 - SIGNAL 3
"A_C41_O4"	Q 1180.7	BOOL	// INTERFACE EXP1 - SIGNAL 4
"A_2145_QXV21_AO1"	QW 168	WORD	// REGULATING VALVE SET POINT
"A_2145_QXV31_AO1"	QW 170	WORD	// REGULATING VALVE SET POINT
"A_2245_QXV21_AO1"	QW 268	WORD	// REGULATING VALVE SET POINT
"A_2245_QXV31_AO1"	QW 270	WORD	// REGULATING VALVE SET POINT
"A_2345_QXV21_AO1"	QW 368	WORD	// REGULATING VALVE SET POINT
"A_2345_QXV31_AO1"	QW 382	WORD	// REGULATING VALVE SET POINT
"A_2445_QXV21_AO1"	QW 468	WORD	// REGULATING VALVE SET POINT
"A_2445_QXV31_AO1"	QW 482	WORD	// REGULATING VALVE SET POINT
"CTUD"	SFB 2	SFB 2	// Count Up / Down
"TON"	SFB 4	SFB 4	// Generate an On Delay
"SIEMENS_BSEND"	SFB 12	SFB 12	// SIEMENS: Block Oriented Send
"SIEMENS_BRCV"	SFB 13	SFB 13	// SIEMENS: Block Oriented Receive
"SIEMENS_HS_COUNT"	SFB 29	SFB 29	// SIEMENS: High-Speed Counter (CPU 312, Integrated Function)
"SIEMENS_FREQ_MES"	SFB 30	SFB 30	// SIEMENS: Frequency Meter (CPU 312, Integrated Function)
"SIEMENS_POSITION"	SFB 31	SFB 31	// SIEMENS: Open-Loop Positioning (CPU 312, Integrated Function)
"SIEMENS_SET_CLK"	SFC 0	SFC 0	// SIEMENS: Set System Clock
"SIEMENS_READ_CLK"	SFC 1	SFC 1	// SIEMENS: Read System Clock
"SIEMENS_SET_RTM"	SFC 2	SFC 2	// SIEMENS: Set Run-Time Meter
"SIEMENS_CTRL_RTM"	SFC 3	SFC 3	// SIEMENS: Start/Stop Run-Time Meter
"SIEMENS_READ_RTM"	SFC 4	SFC 4	// SIEMENS: Read Run-Time Meter
"GADR_LGC"	SFC 5	SFC 5	// Query Logical Address of a Channel
"RD_SINFO"	SFC 6	SFC 6	// Read OB Start Information
"DPNRM_DG"	SFC 13	SFC 13	// Read Diagnostic Data of a DP Slave
"SIEMENS_DPRD_DAT"	SFC 14	SFC 14	// SIEMENS: Read data for DP-Node
"SIEMENS_DPWR_DAT"	SFC 15	SFC 15	// SIEMENS: Write Data to DP-Node
"SIEMENS_BLKMOV"	SFC 20	SFC 20	// SIEMENS: Direct Word Move
"SIEMENS_FILL"	SFC 21	SFC 21	// SIEMENS: Initialize a memory area
"SIEMENS_CREAT_DB"	SFC 22	SFC 22	// SIEMENS: Create Data Block
"SIEMENS_TEST_DB"	SFC 24	SFC 24	// SIEMENS: Test DB
"SIEMENS_SET_TINT"	SFC 28	SFC 28	// SIEMENS: Set Time-of-Day Interrupt
"SIEMENS_CAN_TINT"	SFC 29	SFC 29	// SIEMENS: Cancel Time-of-Day Interrupt
"SIEMENS_ACT_TINT"	SFC 30	SFC 30	// SIEMENS: Activate Time-of-Day Interrupt
"SIEMENS_QRY_TINT"	SFC 31	SFC 31	// SIEMENS: Query Time-of-Day Interrupt
"SIEMENS_SRT_DINT"	SFC 32	SFC 32	// SIEMENS: Start Time-Delay Interrupt
"SIEMENS_CAN_DINT"	SFC 33	SFC 33	// SIEMENS: Cancel Time-Delay Interrupt
"SIEMENS_QRY_DINT"	SFC 34	SFC 34	// SIEMENS: Query Time-Delay Interrupt
"SIEMENS_MSK_FLT"	SFC 36	SFC 36	// SIEMENS: Mask synchronous faults
"SIEMENS_DMSK_FLT"	SFC 37	SFC 37	// SIEMENS: Unmask Synchronous Faults
"SIEMENS_READ_ERR"	SFC 38	SFC 38	// SIEMENS: Read Error Registers
"SIEMENS_DIS_IRT"	SFC 39	SFC 39	// SIEMENS: Disable Interrupt
"SIEMENS_EN_IRT"	SFC 40	SFC 40	// SIEMENS: Enable New Interrupts and Asynchronous Errors
"SIEMENS_DIS_AIRT"	SFC 41	SFC 41	// SIEMENS: Disable Alarm Interrupts
"SIEMENS_EN_AIRT"	SFC 42	SFC 42	// SIEMENS: Enable Alarm Interrupts
"SIEMENS_RE_TRIGR"	SFC 43	SFC 43	// SIEMENS: Retrigger Cycle Time Monitoring
"SIEMENS_REPL_VAL"	SFC 44	SFC 44	// SIEMENS: Replace Value
"SIEMENS_STP"	SFC 46	SFC 46	// SIEMENS: Change the CPU to STOP
"SIEMENS_WAIT"	SFC 47	SFC 47	// SIEMENS: Wait
"SIEMENS_LGC_GADR"	SFC 49	SFC 49	// SIEMENS:
"SIEMENS_RD_LGADR"	SFC 50	SFC 50	// SIEMENS:
"SIEMENS_RDSYSST"	SFC 51	SFC 51	// SIEMENS: Read System Status
"SIEMENS_WR_USMSG"	SFC 52	SFC 52	// SIEMENS: Write User Element in Diagnosis Buffer
"SIEMENS_WR_PARM"	SFC 55	SFC 55	// SIEMENS: Synchronous Write Parameter (MC7)
"SIEMENS_WR_DPARM"	SFC 56	SFC 56	// SIEMENS: Synchronous Write Parameter (SDB)
"SIEMENS_PARM_MOD"	SFC 57	SFC 57	// SIEMENS: Synchronous Write Static and Dynamic
"SIEMENS_WR_REC"	SFC 58	SFC 58	// SIEMENS: Write Data Record
"SIEMENS_RD_REC"	SFC 59	SFC 59	// SIEMENS: Read Data Record
"SIEMENS_AB_CALL"	SFC 63	SFC 63	// SIEMENS: Assembly Code Block (CPU 614)
"SIEMENS_TIME_TCK"	SFC 64	SFC 64	// SIEMENS: Time Tick
"SYS_PLCStartUpDelay"	T 10	TIMER	// SYS: Delay software enable after plc startup
"SYS_HWDelay"	T 11	TIMER	// SYS: Delay software enable after hardware stop
"SYS_T_LOGEntryDelay"	T 13	TIMER	// SYS: Delay log entrys after fuse tripped
"SYS_T_OfflineDelay"	T 14	TIMER	// SYS: Delay section staOffline
"SYS_T_NStartOfflineTime"	T 15	TIMER	// SYS: Offline time after a newstart
"SYS_DelayHeavyStartup"	T 16	TIMER	// SYS: Monitoring time to reset flag
"SYS_DelayBrakeMill"	T 17	TIMER	// SYS: Monitoring time to reset flag brake mill
"COM_T_PCCWatchdog"	T 20	TIMER	// COM: Communication monitoring to process control computer
"SEW_MOVIDRIVE"	UDT 200	UDT 200	// MOVIDRIVE DFP21 (DPV1)
"DANFOSS_VLT5000"	UDT 203	UDT 203	// Danfoss VLT 5000
"ABB_ACS800"	UDT 204	UDT 204	// ABB ACS800 / RPBA-01
"NORDAC"	UDT 205	UDT 205	// NORDAC_SK500_SK TU3-PBR
"ASW_Flags_F0_F15"	UDT 1000	UDT 1000
"ASW_LineAnimation"	UDT 1001	UDT 1001
"ASW_UserSectionState"	UDT 1002	UDT 1002
"ASW_ProductInfo"	UDT 1003	UDT 1003
"SSA_HandAddInfo"	UDT 1004	UDT 1004
"ASW_DFCARecipe"	UDT 1005	UDT 1005
"SSA_MH_ProcessTime"	UDT 2000	UDT 2000	// Malthouse Actual time Process
"SSA_MH_StepTime"	UDT 2001	UDT 2001	// Malthouse Actual time Step
"SSA_MH_JobHeader"	UDT 2003	UDT 2003	// Malthouse SecNom: Job_Header
"SSA_MH_SecNomStandPIC"	UDT 2004	UDT 2004	// Malthouse SecNom: Standard Command PC
"SSA_MH_Step_Loading"	UDT 2011	UDT 2011	// Malthouse Step Loading
"SSA_MH_Step_Unloading"	UDT 2012	UDT 2012	// Malthouse Step Unloading
"SSA_MH_Step_Clearing"	UDT 2013	UDT 2013	// Malthouse Step Clearing
"SSA_Steep_Cmd"	UDT 2100	UDT 2100	// Steeping Section: Commands
"SSA_Steep_Par"	UDT 2101	UDT 2101	// Steeping Section: Parameter
"SSA_Steep_Recipe"	UDT 2102	UDT 2102	// Steeping Section: Recipe
"SSA_Steep_Analog"	UDT 2103	UDT 2103	// Steeping Section: Analog Values
"SSA_Steep_Recipe_Header"	UDT 2104	UDT 2104	// Steeping Section: Recipe Header
"SSA_Steep_Step"	UDT 2105	UDT 2105	// Steeping Section : Single Step
"SSA_Steep_Sum"	UDT 2106	UDT 2106	// Summary values for Steeping with sequencial conical steep
"SSA_Germ_Cmd"	UDT 2200	UDT 2200	// Germination Section: Commands
"SSA_Germ_Par"	UDT 2201	UDT 2201	// Germination Section: Parameter
"SSA_Germ_Recipe"	UDT 2202	UDT 2202	// Germination Section: Recipe
"SSA_Germ_Analog"	UDT 2203	UDT 2203	// Germination Section: Analog Values
"SSA_Germ_Recipe_Header"	UDT 2204	UDT 2204	// Germination Section:  Recipe Header
"SSA_Germ_Step"	UDT 2205	UDT 2205	// Germination Section: Single Step
"SSA_Kiln_Cmd"	UDT 2300	UDT 2300	// Kilning Section: Commands
"SSA_Kiln_Par"	UDT 2301	UDT 2301	// Kilning Section: Parameter
"SSA_Kiln_Recipe"	UDT 2302	UDT 2302	// Kilning Section: Recipe
"SSA_Kiln_Analog"	UDT 2303	UDT 2303	// Kilning Section: Analog Values
"SSA_Kiln_Recipe_Header"	UDT 2304	UDT 2304	// Kilning Section:  Recipe Header
"SSA_Kiln_Step"	UDT 2305	UDT 2305	// Kilning Section: Single Step
"UDTL01LineCmd"	UDT 3200	UDT 3200
"UDTL01SecData"	UDT 3202	UDT 3202
"UDTL01SecAc"	UDT 3203	UDT 3203
"UDTL01SecNom"	UDT 3204	UDT 3204
"ASW_DEC1OnOffCmd"	UDT 5000	UDT 5000	// ASW: Line Command
"ASW_DEC1SecNom"	UDT 5001	UDT 5001	// ASW: Nominal Data
"ASW_DEC1SecAc"	UDT 5002	UDT 5002	// ASW: Actual Data
"ASW_EXP1OnOffCmd"	UDT 5100	UDT 5100	// ASW: Line Command
"ASW_EXP1SecNom"	UDT 5101	UDT 5101	// ASW: Nominal Data
"ASW_EXP1SecAc"	UDT 5102	UDT 5102	// ASW: Actual Data
"ASW_MAL1OnOffCmd"	UDT 8000	UDT 8000	// ASW: Line Command
"ASW_MAL1SecNom"	UDT 8001	UDT 8001	// ASW: Nominal Data
"ASW_MAL1SecAc"	UDT 8002	UDT 8002	// ASW: Actual Data
"CMDs_ILO_Funktion"	UDT 8015	UDT 8015	// Command and setpoints for one ILO-funktion
"SSA_LOG_Value"	UDT 10005	UDT 10005
"ASW_CBitDeclaration"	UDT 10020	UDT 10020	// ASW: Declaration of change bit data blocks
"GCS7_UDT_Timer"	UDT 10180	UDT 10180	// Timer in DB
"CWA_UDT_Command"	UDT 10413	UDT 10413	// UDT Command  for CWA
"CWA_UDT_BinParaShort"	UDT 10418	UDT 10418	// UDT CWA bin parameter with minimum used parameter
"CWA_UDT_BinParaAll"	UDT 10419	UDT 10419	// UDT CWA bin parameter with all parameters
"GCS7_UDT_FunctionKey"	UDT 10601	UDT 10601	// GCS7: Upper Layer
"GCS7_UDT_FaultPattern"	UDT 10602	UDT 10602	// GCS7: Upper Layer
"GCS7_UDT_StatusPattern"	UDT 10603	UDT 10603	// Upper Layer
"GCS7_UDT_BINList1"	UDT 10660	UDT 10660	// GCS7: Binlist without WtActual and WtTarget
"GCS7_UDT_BINStatus"	UDT 10662	UDT 10662	// GCS7: Binstatus
"GCS7_UDT_BINList2"	UDT 10664	UDT 10664	// GCS7: Binlist with WtActual without WtTarget
"GCS7_UDT_BINList3"	UDT 10668	UDT 10668	// GCS7: Binlist with WtActual and WtTarget
"GCS7_UDT_ScaleControl"	UDT 10680	UDT 10680	// GCS7: Scale control
"ASW_StageCtrl"	UDT 18000	UDT 18000
"PCCYieldScale"	UDT 19000	UDT 19000	// USW: Struct for scales involved in yield calculation
"WinCoSYieldScale"	UDT 19001	UDT 19001	// USW: Struct for scales involved in yield calculation
"SamplerData"	UDT 19002	UDT 19002	// USW: Struct for sampler data
"BigBagData"	UDT 19003	UDT 19003	// Registration of big bag weight
"GCS7_FB9_Section"	UDT 20090	UDT 20090	// Group Control: Interface Section
"GCS7_GR_COM"	UDT 20097	UDT 20097	// GCS7 Data PLC Communication per group
"GCS90S7_FB9_Communicat"	UDT 20098	UDT 20098	// Communication PLC --PLC GCS7 to GCS90S7
"GCS7_FB9_Communication"	UDT 20099	UDT 20099	// Communication PLC --PLC
"GCS7_FB11_Communication"	UDT 20119	UDT 20119	// Communication PLC --PLC
"GCS7_FB12_Communication"	UDT 20129	UDT 20129	// Communication PLC --PLC
"GCS7_FB13_Communication"	UDT 20139	UDT 20139	// Communication PLC --PLC
"GCS7_FB14_Communication"	UDT 20149	UDT 20149	// Communication PLC --PLC
"GCS7_FB16_Communication"	UDT 20169	UDT 20169	// Communication PLC --PLC
"GCS7_FB37_DP_Alarm"	UDT 20373	UDT 20373	// SSW: Element MDDR/T Alarms
"GCS7_FB40_dynData"	UDT 20400	UDT 20400	// Lower Layer
"GCS7_M_FB41_Data"	UDT 20410	UDT 20410	// Lower Layer
"GCS7_M_FB44_Data"	UDT 20440	UDT 20440	// Lower Layer
"GCS7_M_FB45_Data"	UDT 20450	UDT 20450	// Lower Layer
"GCS7_M_FB46_Data"	UDT 20460	UDT 20460	// Lower Layer
"GCS7_M_FB47_Data"	UDT 20470	UDT 20470	// Lower Layer
"GCS7_M_FB48_Data"	UDT 20480	UDT 20480	// Lower Layer
"GCS7_M_FB49_Data"	UDT 20490	UDT 20490	// Lower Layer
"GCS7_M_FB50_Data"	UDT 20500	UDT 20500	// Lower Layer
"GCS7_M_FB51_Data"	UDT 20510	UDT 20510	// Lower Layer
"GCS7_M_FB52_Data"	UDT 20520	UDT 20520	// Lower Layer
"GCS7_M_FB53_Data"	UDT 20530	UDT 20530	// Lower Layer
"GCS7_M_FB54_Data"	UDT 20540	UDT 20540	// Lower Layer
"GCS7_M_FB55_Data"	UDT 20550	UDT 20550	// Lower Layer
"GCS7_M_FB56_Data"	UDT 20560	UDT 20560	// Lower Layer
"GCS7_M_FB58_Data"	UDT 20580	UDT 20580	// Lower Layer
"GCS7_M_FB59_Data"	UDT 20590	UDT 20590	// Lower Layer
"GCS7_M_FB60_Data"	UDT 20600	UDT 20600	// Lower Layer
"GCS7_M_FB61_Data"	UDT 20610	UDT 20610	// Lower Layer
"GCS7_M_FB62_Data"	UDT 20620	UDT 20620	// Lower Layer
"GCS7_M_FB63_Data"	UDT 20630	UDT 20630	// Lower Layer
"GCS7_M_FB64_Data"	UDT 20640	UDT 20640	// Lower Layer
"GCS7_M_FB65_Data"	UDT 20650	UDT 20650	// Lower Layer
"GCS7_M_FB66_Data"	UDT 20660	UDT 20660	// Lower Layer
"GCS7_M_FB67_Data"	UDT 20670	UDT 20670	// Lower Layer
"GCS7_M_FB68_Data"	UDT 20680	UDT 20680	// Lower Layer
"GCS7_M_FB69_Data"	UDT 20690	UDT 20690	// Lower Layer
"GCS7_E_FB73_A201"	UDT 20735	UDT 20735	// DFCA: Data Telegram A201:
"GCS7_M_FB81_Data"	UDT 20810	UDT 20810	// Lower Layer
"GCS7_M_FB82_Data"	UDT 20820	UDT 20820	// Lower Layer
"GCS7_FB84_Communication"	UDT 20849	UDT 20849	// Communication PLC --PLC
"GCS7_FB85_Data"	UDT 20850	UDT 20850	// Stroke Drive
"GCS7_FB85_Counter"	UDT 20851	UDT 20851	// Data of Increment counter
"GCS7_FB86_Data"	UDT 20860	UDT 20860
"GCS7_FB87_Data"	UDT 20861	UDT 20861
"GCS7_M_FB87_Data"	UDT 20870	UDT 20870	// Machine 4/8 roll stand with profibus
"GCS7_M_FB88_Data"	UDT 20880	UDT 20880	// Machin Flat-bottom discharger
"GR052_UDT"	UDT 21520	UDT 21520	// UDT way groupAspiration Flaps Bin 21 to 34 (Aspiration)
"G282M_UDT"	UDT 23820	UDT 23820	// UDT way groupFLAP BOX 9008
"G314W_UDT"	UDT 24140	UDT 24140	// UDT way groupSLIDES UNDER CHAIN CONV. 6118
"G316W_UDT"	UDT 24160	UDT 24160	// UDT way groupSLIDES UNDER CHAIN CONV. 6113
"G317W_UDT"	UDT 24170	UDT 24170	// UDT way groupOUTLET SLIDES MALT BUFFER BINS
"SSW_EL_ASI_Slave"	UDT 28995	UDT 28995	// Element Control ASI Master Wago/Profibus Slave Data
"ASW_UDTOnOffCmd"	UDT 32700	UDT 32700
"ASW_UDTSecNom"	UDT 32701	UDT 32701	// Nominal value for section
"ASW_UDTSecAc"	UDT 32702	UDT 32702	// Actual values of section
"VAT_Sections_Kom_5_7"	VAT 1	
"I/O Check"	VAT 2		// I/O Check
"VAT_KK1_Count"	VAT 3	
"VAT_D1_D2_Count"	VAT 4	
"vat_donk1"	VAT 6	
"VAT_MERKERS_RESET_FC"	VAT 7	
"VAT_vent_connections"	VAT 8	
"VAT_vent_asdasd"	VAT 9	
"VAT_CBitDB1005"	VAT 15	
END_SYMBOL_TABLE

